// SIMATIC STEP 7 (V5.x) project Mangal
// CPU: CPU 416-2 DP
// station: Hardware
// station: SIMATIC 400
// station: P_ADR_BUS
// program: S7 Program(1)

SYMBOL_TABLE
"CONT_C"	FB 1	FB 1	// Continuous PID controller
"TIMER_P"	FB 5	FB 5	// Impulsefunction and delayed On/Off
"RAMP_P"	FB 52	FB 52
"N_PID"	FB 55	FB 55
"regulator"	FB 321	FB 321
"CBCTRLS1"	FB 945	FB 945	// CB SEND DATA 1 TO CTR
"VISU_IND_CODE"	FB 982	FB 982	// VISU COLOR INDICATION CODE
"READY_STD"	FB 1060	FB 1060	// Diagnosis  block
"VISU_GEN"	FB 1067	FB 1067	// Visualisierung for general Indications
"N_AnMeas"	FB 1435	FB 1435
"N_SPMANIP"	FB 1467	FB 1467
"N_TON"	FB 1482	FB 1482
"N_TOF"	FB 1483	FB 1483
"CUT_SHER"	FB 3333	FB 3333
"A_IN"	FC 402	FC 402	// Analog Input Driver
"N_AW_BO"	FC 430	FC 430
"CYCL_EXC"	OB 1	OB 1	// Cycle Execution
"PROG_ERR"	OB 121	OB 121	// Programming Error
"MOD_ERR"	OB 122	OB 122	// Module Access Error
"TON"	SFB 4	SFB 4	// Generate an On Delay
"TOF"	SFB 5	SFB 5	// Generate an Off Delay
"ALARM_8P"	SFB 35	SFB 35	// Generate Block-Related Messages with Values for 8 Signals
"RD_SINFO"	SFC 6	SFC 6	// Read OB Start Information
"BLKMOV"	SFC 20	SFC 20	// Copy Variables
"TIME_TCK"	SFC 64	SFC 64	// Read the System Time
END_SYMBOL_TABLE

FUNCTION_BLOCK "CONT_C"	// FB 1
TITLE = Continuous PID controller
AUTHOR : ELEM_400
FAMILY : CONTROL
NAME : CONT_C
VERSION : 1.5
VAR_INPUT
  MAN_ON : BOOL  := TRUE;	//Select: 1=Manual Value, 0= Manip. Value
  PVPER_ON { S7_visible := 'false' }: BOOL ;	//Enable: 1=Process var. to Peripherl Dev.
  P_SEL : BOOL  := TRUE;	//1=Proportional Action ON
  I_SEL : BOOL  := TRUE;	//Enable: 1=Integral Action ON
  INT_HOLD : BOOL ;	//Integral Action Hold
  I_ITL_ON : BOOL ;	//Initialize Integral Action
  D_SEL : BOOL ;	//1=Derivative Action ON
  SAMPLE_T { S7_visible := 'false'; S7_sampletime := 'true' }: REAL  := 1.000000e+000;	//Sample Time [s]
  SP_INT : REAL ;	//Internal setpoint
  PV_IN { S7_dynamic := 'true' }: REAL ;	//Process Variable Input
  PV_PER : WORD ;	//Process Variable from Peripheral Device
  MAN : REAL ;	//Operator Entered Manual Value
  GAIN { S7_dynamic := 'true'; S7_edit := 'para' }: REAL  := 2.000000e+000;	//Proportional Gain
  TN { S7_dynamic := 'true'; S7_edit := 'para' }: TIME  := T#20S;	//Reset time [sec]
  TV { S7_dynamic := 'true'; S7_edit := 'para' }: TIME  := T#10S;	//Differential Time [s]
  TM_LAG : TIME  := T#2S;	//Lag Time of the Derivative Action [sec]
  DEADB_W : REAL ;	//Deadband width
  LMN_HLM : REAL  := 1.000000e+002;	//Manipulated Value High Limit
  LMN_LLM : REAL ;	//Manipulated Value Low Limit
  PV_FAC { S7_visible := 'false' }: REAL  := 1.000000e+000;	//Process Variable Adjustment Factor
  PV_OFF { S7_visible := 'false' }: REAL ;	//Process Variable Offset
  LMN_FAC : REAL  := 1.000000e+000;	//Manipulated Value Adjustment Factor
  LMN_OFF : REAL ;	//Manipulated Value Offset
  I_ITLVAL : REAL ;	//Initialization Value of Integral Action
  DISV : REAL ;	//Disturbance variable
END_VAR
VAR_OUTPUT
  LMN : REAL ;	//Manipulated Value
  LMN_PER : WORD ;	//Manipulated Value for Peripheral Device
  QLMN_HLM : BOOL ;	//1=High Limit of Manipulated Value active
  QLMN_LLM : BOOL ;	//1=Low Limit of Manipulated Value active
  LMN_P : REAL ;	//Proportionality Component
  LMN_I : REAL ;	//Integral Component
  LMN_D : REAL ;	//Derivative Component
  PV { S7_visible := 'false' }: REAL ;	//Process Variable
  ER : REAL ;	//Error Signal
END_VAR
VAR
  sInvAlt : REAL ;
  sIanteilAlt : REAL ;
  sRestInt : REAL ;
  sRestDif : REAL ;
  sRueck : REAL ;
  sLmn : REAL ;
  sbArwHLmOn : BOOL ;
  sbArwLLmOn : BOOL ;
  sbILimOn : BOOL  := TRUE;
END_VAR
VAR_TEMP
  ERR : INT ;
  TOP_SI : STRUCT
   EV_CLASS : BYTE ;
   EV_NUM : BYTE ;
   PRIORITY : BYTE ;
   NUM : BYTE ;
   TYP2_3 : BYTE ;
   TYP1 : BYTE ;
   ZI1 : WORD ;
   ZI2_3 : DWORD ;
  END_STRUCT ;
  START_UP_SI : STRUCT
   EV_CLASS : BYTE ;
   EV_NUM : BYTE ;
   PRIORITY : BYTE ;
   NUM : BYTE ;
   TYP2_3 : BYTE ;
   TYP1 : BYTE ;
   ZI1 : WORD ;
   ZI2_3 : DWORD ;
  END_STRUCT ;
  Hvar : REAL ;	//Hilfsvariable
  Diff : REAL ;	//Änderungswert
  Istwert : REAL ;	//Istwert
  ErKp : REAL ;	//Hilfsvariable
  rTi : REAL ;	//Integrationszeit in real
  rTd : REAL ;	//Differentiationszeit in real
  rTmLag : REAL ;	//Verzögerungszeit in real
  Panteil : REAL ;	//P-Anteil
  Ianteil : REAL ;	//I-Anteil
  Danteil : REAL ;	//D-Anteil
  Verstaerk : REAL ;	//Verstärkung
  RueckDiff : REAL ;	//Differenz des Rückkopplungswertes
  RueckAlt : REAL ;	//Alter Rückkopplungswert
  dLmn : REAL ;	//Stellwert
  gf : REAL ;	//Hilfwert
  rVal : REAL ;	//Real Hilfsvariable
END_VAR
BEGIN
// body was compiled from an SCL source; compiled code not shown
END_FUNCTION_BLOCK

// FB 5: know-how protected block, not included

FUNCTION_BLOCK FB 45
VERSION : 0.1
BEGIN
// (block stored without names or comments; labels and parameter names are numbered)
END_FUNCTION_BLOCK

FUNCTION_BLOCK "RAMP_P"	// FB 52
TITLE = Rampforming
AUTHOR : BASIS70
FAMILY : CONTROL
NAME : RAMP_P
VERSION : 3.0
VAR_INPUT
  SAMPLE_T { S7_visible := 'false'; S7_sampletime := 'true' }: REAL  := 1.000000e+000;	//Sample Time [s]
  URLM { S7_dynamic := 'true'; S7_edit := 'para' }: REAL  := 3.000000e+000;	//Positive Ramp Rate Limit Output Value
  DRLM { S7_dynamic := 'true'; S7_edit := 'para' }: REAL  := 3.000000e+000;	//Max. negative Ramp Rate of Output Value
  U { S7_dynamic := 'true' }: REAL ;	//Input Value
  RATE_OFF { S7_dynamic := 'true' }: BOOL ;	//1=Ramp Rate Monitoring off
END_VAR
VAR_OUTPUT
  QERR { S7_visible := 'false' }: BOOL  := TRUE;	//1=Error
  QLIM_U { S7_dynamic := 'true' }: BOOL ;	//1=Positiv Ramp Rate Limit Active
  QLIM_D { S7_dynamic := 'true' }: BOOL ;	//1=Negativ Ramp Rate Limit Active
  V { S7_dynamic := 'true' }: REAL ;	//Analog Output
END_VAR
VAR
  srSAMPLE_T : REAL ;	//interne Abtastzeit
END_VAR
VAR_TEMP
  tbQlim_u : BOOL ;	//Hilfsmerker positiver Gradient zu gross
  tbQlim_d : BOOL ;	//Hilfsmerker negativer Gradient zu gross
  trGrad : REAL ;	//Gradient
  trDiff : REAL ;	//temporäre Var. für U-V
  ERR : INT ;	//Error beim Anlauf
  TOP_SI : STRUCT
   EV_CLASS : BYTE ;
   EV_NUM : BYTE ;
   PRIORITY : BYTE ;
   NUM : BYTE ;
   TYP2_3 : BYTE ;
   TYP1 : BYTE ;
   ZI1 : WORD ;
   ZI2_3 : DWORD ;
  END_STRUCT ;
  START_UP_SI : STRUCT
   EV_CLASS : BYTE ;
   EV_NUM : BYTE ;
   PRIORITY : BYTE ;
   NUM : BYTE ;
   TYP2_3 : BYTE ;
   TYP1 : BYTE ;
   ZI1 : WORD ;
   ZI2_3 : DWORD ;
  END_STRUCT ;
END_VAR
BEGIN
// body was compiled from an SCL source; compiled code not shown
END_FUNCTION_BLOCK

FUNCTION_BLOCK "N_PID"	// FB 55
VERSION : 0.1
VAR_INPUT
  PLCAUTOSP : BOOL ;
  PLCMANSP : BOOL ;
  PLCAUTOPOS : BOOL ;
  PLCMANPOS : BOOL ;
  P_SEL { S7_m_c := 'true' }: BOOL ;
  I_SEL { S7_m_c := 'true' }: BOOL ;
  D_SEL { S7_m_c := 'true' }: BOOL ;
  INT_HOLD : BOOL ;
  INT_INIT : BOOL ;
  SPAUTO { S7_m_c := 'true' }: REAL ;
  SPAUTOPOS { S7_m_c := 'true' }: REAL ;
  PV { S7_m_c := 'true' }: REAL ;
  GAIN { S7_m_c := 'true'; S7_dynamic := 'true' }: REAL ;
  TN { S7_dynamic := 'true'; S7_m_c := 'true' }: REAL ;
  TV { S7_dynamic := 'true'; S7_m_c := 'true' }: REAL ;
  TM_LAG : REAL ;
  DEAD_W : REAL ;
  DEV { S7_dynamic := 'true'; S7_m_c := 'true' }: REAL ;
  DEV_TIME { S7_dynamic := 'true'; S7_m_c := 'true' }: REAL ;	//Deviation time [s]
  LNM_HLIM : REAL ;
  LNM_LLIM : REAL ;
  I_INITVAL : REAL ;
  DISV : REAL ;
  SAMPLE_T { S7_sampletime := 'true' }: REAL ;
END_VAR
VAR_OUTPUT
  QAUTOSP { S7_dynamic := 'true'; S7_m_c := 'true' }: BOOL ;
  QMANSP { S7_dynamic := 'true'; S7_m_c := 'true' }: BOOL ;
  QAUTOPOS { S7_dynamic := 'true'; S7_m_c := 'true' }: BOOL ;
  QMANPOS { S7_dynamic := 'true'; S7_m_c := 'true' }: BOOL ;
  QLMN { S7_dynamic := 'true'; S7_m_c := 'true' }: REAL ;
  QLMN_P : REAL ;
  QLMN_I : REAL ;
  QLMN_D : REAL ;
  QLMN_HLIM : BOOL ;
  QLMM_LLIM : BOOL ;
  QDEV_H { S7_m_c := 'true' }: BOOL ;
  QDEV_L { S7_m_c := 'true' }: BOOL ;
  QDEV : BOOL ;
  QDEV_ACT : REAL ;
  QPID_SP { S7_dynamic := 'true'; S7_m_c := 'true' }: REAL ;
  QER { S7_dynamic := 'true'; S7_m_c := 'true' }: REAL ;
END_VAR
VAR_IN_OUT
  HMIAUTOSP { S7_dynamic := 'true'; S7_m_c := 'true' }: BOOL ;
  HMIMANSP { S7_dynamic := 'true'; S7_m_c := 'true' }: BOOL ;
  HMIAUTOPOS { S7_dynamic := 'true'; S7_m_c := 'true' }: BOOL ;
  HMIMANPOS { S7_dynamic := 'true'; S7_m_c := 'true' }: BOOL ;
  HMISPMAN { S7_dynamic := 'true'; S7_m_c := 'true' }: REAL ;
  HMISPMANPOS { S7_dynamic := 'true'; S7_m_c := 'true' }: REAL ;
  HMIOPEN { S7_m_c := 'true' }: BOOL ;
  HMICLOSE { S7_m_c := 'true' }: BOOL ;
END_VAR
VAR
  AutoSPMode_Int : BOOL ;
  AutoPosMode_Int : BOOL ;
  ManSPMode_Int : BOOL ;
  ManPosMode_Int : BOOL ;
  Pos : BOOL ;
  Reg : BOOL ;
  Deviation : BOOL ;
  Dev_H : BOOL ;
  Dev_L : BOOL ;
  HMIAtuoSPReq : BOOL ;
  HMIManSPReq : BOOL ;
  HMIAtuoPosReq : BOOL ;
  HMIManPosReq : BOOL ;
  ReqAutoSP : BOOL ;
  ReqManSP : BOOL ;
  ReqAutoPos : BOOL ;
  ReqManPos : BOOL ;
  PulsePLCAutoSP : BOOL ;
  PulsePLCManSP : BOOL ;
  PulsePLCAutoPos : BOOL ;
  PulsePLCManPos : BOOL ;
  Spare_11 : BOOL ;
  Spare_10 : BOOL ;
  Spare_9 : BOOL ;
  Spare_8 : BOOL ;
  Spare_7 : BOOL ;
  Spare_6 : BOOL ;
  Spare_5 : BOOL ;
  Spare_4 : BOOL ;
  Spare_3 : BOOL ;
  Spare_2 : BOOL ;
  Spare_1 : BOOL ;
  Spare1 : REAL ;
  Spare2 : REAL ;
  Spare3 : REAL ;
  AutoSP_Int : REAL ;
  ManSP_Int : REAL ;
  AutoPosSP_Int : REAL ;
  ManPosSP_Int : REAL ;
  PID_SP : REAL ;
  PID_SP_Ramped : REAL ;
  PID_Pos_SP : REAL ;
  PID_Pos_SP_Ramped : REAL ;
  PID_LMN : REAL ;
  Err_Val : REAL ;
  Dev_Val_Abs : REAL ;
  DEV_Act_Int : REAL ;
  DEV_Proc : REAL ;
  Dev_Tmr : SFB 4;
  PID_CTRL : FB 1;
  SP_RAMP : FB 52;
  POS_RAMP : FB 52;
  MANIP_SP : FB 1467;
END_VAR
VAR_TEMP
  Log_1 : BOOL ;
  Log_0 : BOOL ;
  TN_Int : TIME ;
  TV_Int : TIME ;
  TM_LAG_Int : TIME ;
  Dev_Time_Int : TIME ;
  Temp_Real : REAL ;
  Dummy_S5 : BOOL ;
END_VAR
BEGIN
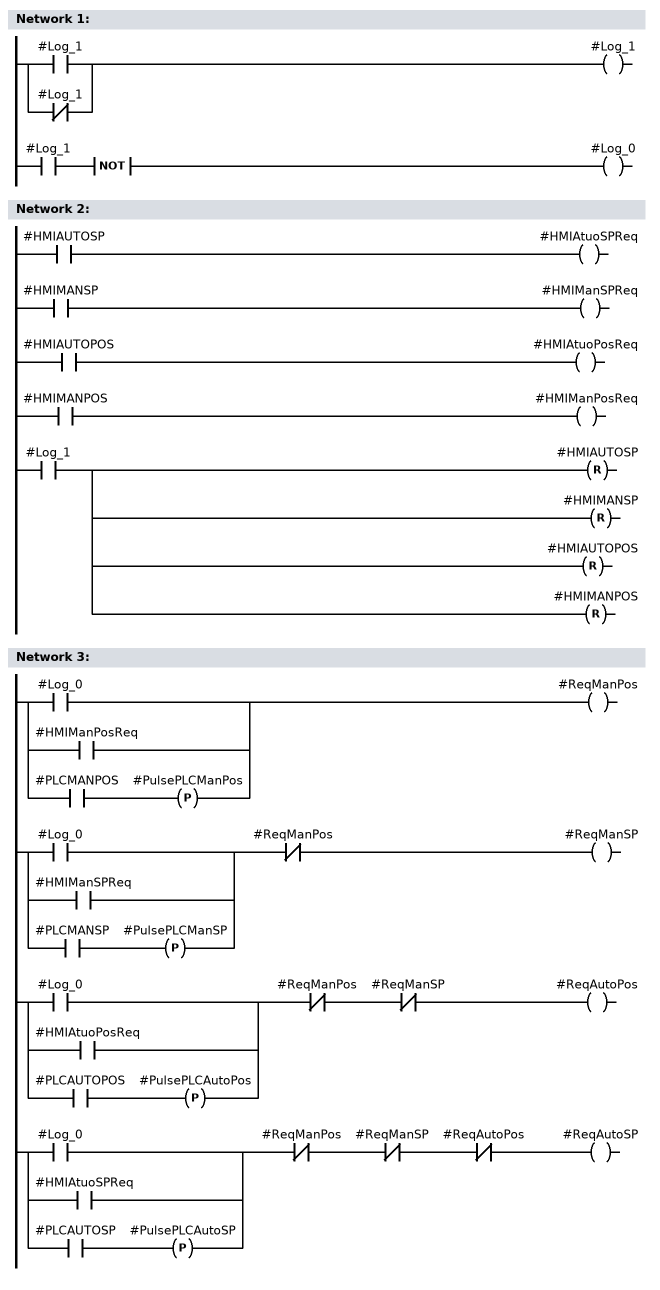
NETWORK
TITLE =
      A(;
      O     #Log_1;
      ON    #Log_1;
      );
      =     #Log_1;
      A     #Log_1;
      NOT;
      =     #Log_0;
NETWORK
TITLE =
      A     #HMIAUTOSP;
      =     #HMIAtuoSPReq;
      A     #HMIMANSP;
      =     #HMIManSPReq;
      A     #HMIAUTOPOS;
      =     #HMIAtuoPosReq;
      A     #HMIMANPOS;
      =     #HMIManPosReq;
      A     #Log_1;
      R     #HMIAUTOSP;
      R     #HMIMANSP;
      R     #HMIAUTOPOS;
      R     #HMIMANPOS;
NETWORK
TITLE =
      A     #Log_0;
      =     L 23.0;
      O     L 23.0;
      O     #HMIManPosReq;
      O(;
      A     #PLCMANPOS;
      FP    #PulsePLCManPos;
      );
      =     #ReqManPos;
      A(;
      O     L 23.0;
      O     #HMIManSPReq;
      O(;
      A     #PLCMANSP;
      FP    #PulsePLCManSP;
      );
      );
      AN    #ReqManPos;
      =     #ReqManSP;
      A(;
      O     L 23.0;
      O     #HMIAtuoPosReq;
      O(;
      A     #PLCAUTOPOS;
      FP    #PulsePLCAutoPos;
      );
      );
      AN    #ReqManPos;
      AN    #ReqManSP;
      =     #ReqAutoPos;
      A(;
      O     L 23.0;
      O     #HMIAtuoSPReq;
      O(;
      A     #PLCAUTOSP;
      FP    #PulsePLCAutoSP;
      );
      );
      AN    #ReqManPos;
      AN    #ReqManSP;
      AN    #ReqAutoPos;
      =     #ReqAutoSP;
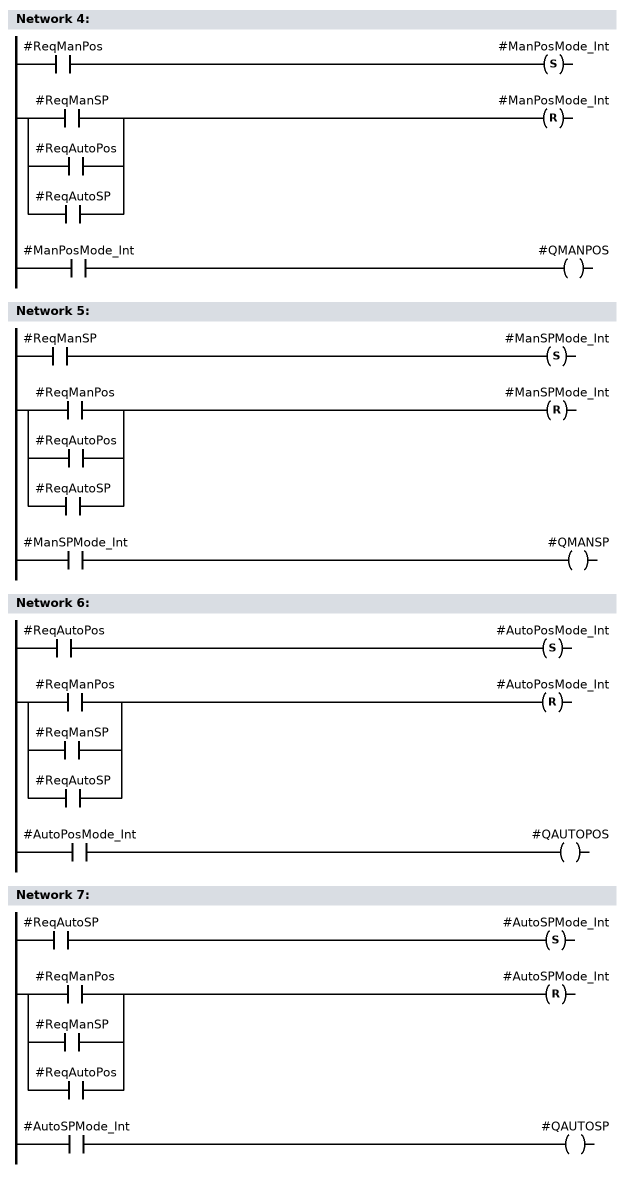
NETWORK
TITLE =
      A     #ReqManPos;
      S     #ManPosMode_Int;
      A(;
      O     #ReqManSP;
      O     #ReqAutoPos;
      O     #ReqAutoSP;
      );
      R     #ManPosMode_Int;
      A     #ManPosMode_Int;
      =     #QMANPOS;
NETWORK
TITLE =
      A     #ReqManSP;
      S     #ManSPMode_Int;
      A(;
      O     #ReqManPos;
      O     #ReqAutoPos;
      O     #ReqAutoSP;
      );
      R     #ManSPMode_Int;
      A     #ManSPMode_Int;
      =     #QMANSP;
NETWORK
TITLE =
      A     #ReqAutoPos;
      S     #AutoPosMode_Int;
      A(;
      O     #ReqManPos;
      O     #ReqManSP;
      O     #ReqAutoSP;
      );
      R     #AutoPosMode_Int;
      A     #AutoPosMode_Int;
      =     #QAUTOPOS;
NETWORK
TITLE =
      A     #ReqAutoSP;
      S     #AutoSPMode_Int;
      A(;
      O     #ReqManPos;
      O     #ReqManSP;
      O     #ReqAutoPos;
      );
      R     #AutoSPMode_Int;
      A     #AutoSPMode_Int;
      =     #QAUTOSP;
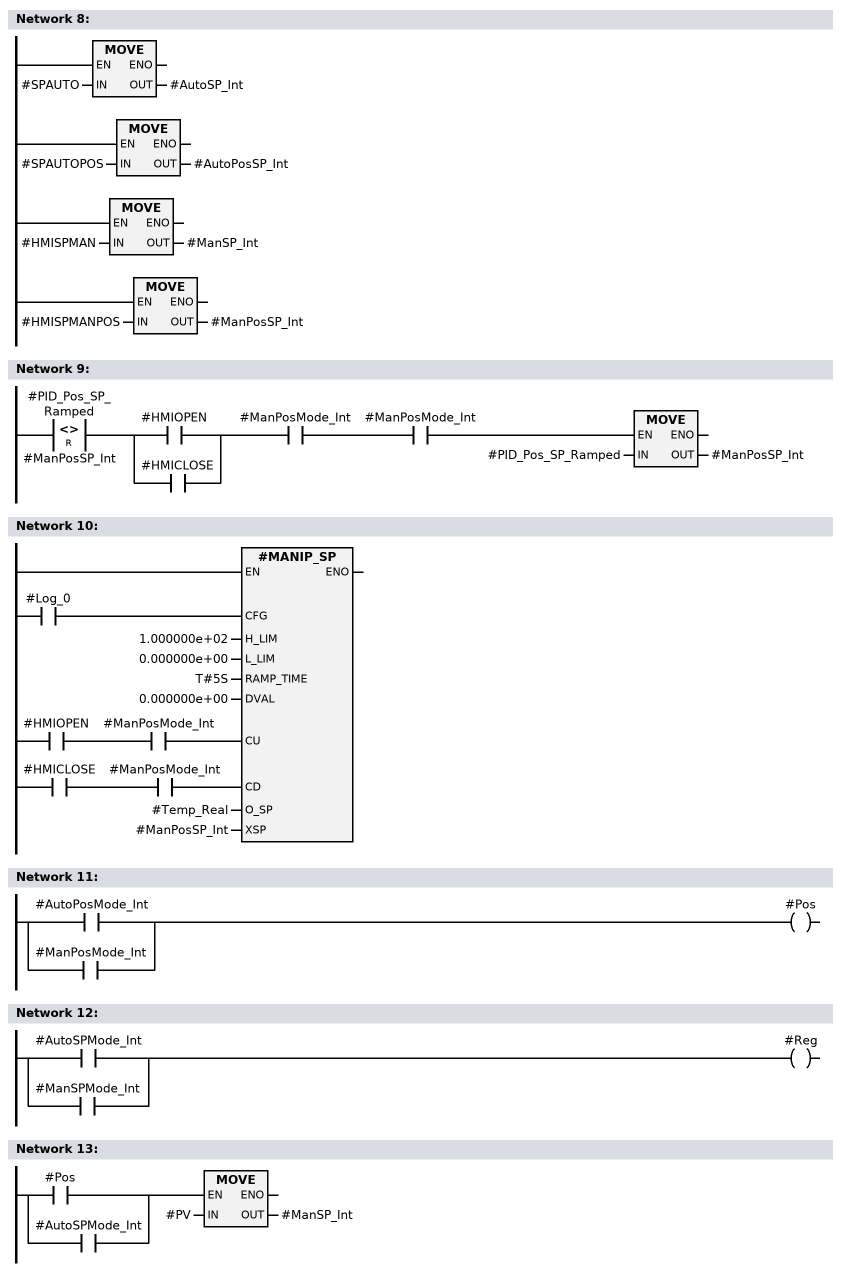
NETWORK
TITLE =
      L     #SPAUTO;
      T     #AutoSP_Int;
      L     #SPAUTOPOS;
      T     #AutoPosSP_Int;
      L     #HMISPMAN;
      T     #ManSP_Int;
      L     #HMISPMANPOS;
      T     #ManPosSP_Int;
NETWORK
TITLE =
      A(;
      L     #PID_Pos_SP_Ramped;
      L     #ManPosSP_Int;
      <>R;
      );
      A(;
      O     #HMIOPEN;
      O     #HMICLOSE;
      );
      A     #ManPosMode_Int;
      A     #ManPosMode_Int;
      JNB   _010;
      L     #PID_Pos_SP_Ramped;
      T     #ManPosSP_Int;
_010: NOP   0;
NETWORK
TITLE =
      A     #Log_0;
      =     L 23.0;
      BLD   103;
      A     #HMIOPEN;
      A     #ManPosMode_Int;
      =     L 23.3;
      BLD   103;
      A     #HMICLOSE;
      A     #ManPosMode_Int;
      =     L 23.4;
      BLD   103;
      CALL  #MANIP_SP (
           CFG                      := L 23.0,
           H_LIM                    := 1.000000e+02,
           L_LIM                    := 0.000000e+00,
           RAMP_TIME                := T#5S,
           DVAL                     := 0.000000e+00,
           CU                       := L 23.3,
           CD                       := L 23.4,
           O_SP                     := #Temp_Real,
           XSP                      := #ManPosSP_Int);
      NOP   0;
NETWORK
TITLE =
      O     #AutoPosMode_Int;
      O     #ManPosMode_Int;
      =     #Pos;
NETWORK
TITLE =
      O     #AutoSPMode_Int;
      O     #ManSPMode_Int;
      =     #Reg;
NETWORK
TITLE =
      A(;
      O     #Pos;
      O     #AutoSPMode_Int;
      );
      JNB   _011;
      L     #PV;
      T     #ManSP_Int;
_011: NOP   0;
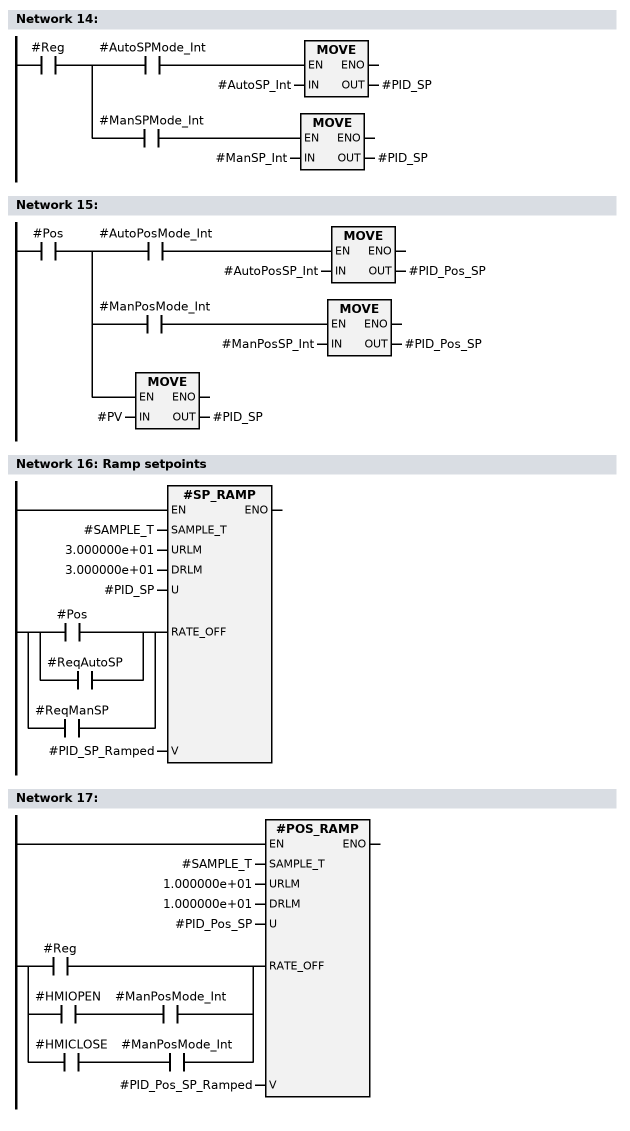
NETWORK
TITLE =
      A     #Reg;
      =     L 23.0;
      A     L 23.0;
      A     #AutoSPMode_Int;
      JNB   _012;
      L     #AutoSP_Int;
      T     #PID_SP;
_012: NOP   0;
      A     L 23.0;
      A     #ManSPMode_Int;
      JNB   _013;
      L     #ManSP_Int;
      T     #PID_SP;
_013: NOP   0;
NETWORK
TITLE =
      A     #Pos;
      =     L 23.0;
      A     L 23.0;
      A     #AutoPosMode_Int;
      JNB   _014;
      L     #AutoPosSP_Int;
      T     #PID_Pos_SP;
_014: NOP   0;
      A     L 23.0;
      A     #ManPosMode_Int;
      JNB   _015;
      L     #ManPosSP_Int;
      T     #PID_Pos_SP;
_015: NOP   0;
      A     L 23.0;
      JNB   _016;
      L     #PV;
      T     #PID_SP;
_016: NOP   0;
NETWORK
TITLE = Ramp setpoints
      A(;
      O     #Pos;
      O     #ReqAutoSP;
      O     #ReqManSP;
      );
      =     L 23.0;
      BLD   103;
      CALL  #SP_RAMP (
           SAMPLE_T                 := #SAMPLE_T,
           URLM                     := 3.000000e+01,
           DRLM                     := 3.000000e+01,
           U                        := #PID_SP,
           RATE_OFF                 := L 23.0,
           V                        := #PID_SP_Ramped);
      NOP   0;
NETWORK
TITLE =
      A(;
      O     #Reg;
      O;
      A     #HMIOPEN;
      A     #ManPosMode_Int;
      O;
      A     #HMICLOSE;
      A     #ManPosMode_Int;
      );
      =     L 23.0;
      BLD   103;
      CALL  #POS_RAMP (
           SAMPLE_T                 := #SAMPLE_T,
           URLM                     := 1.000000e+01,
           DRLM                     := 1.000000e+01,
           U                        := #PID_Pos_SP,
           RATE_OFF                 := L 23.0,
           V                        := #PID_Pos_SP_Ramped);
      NOP   0;
NETWORK
TITLE = Real to TIME conversion
      L     #TN;
      L     1.000000e+03;
      *R;
      RND;
      T     #TN_Int;
      L     #TV;
      L     1.000000e+03;
      *R;
      RND;
      T     #TV_Int;
      L     #TM_LAG;
      L     1.000000e+03;
      *R;
      RND;
      T     #TM_LAG_Int;
      L     #DEV_TIME;
      L     1.000000e+03;
      *R;
      RND;
      T     #Dev_Time_Int;
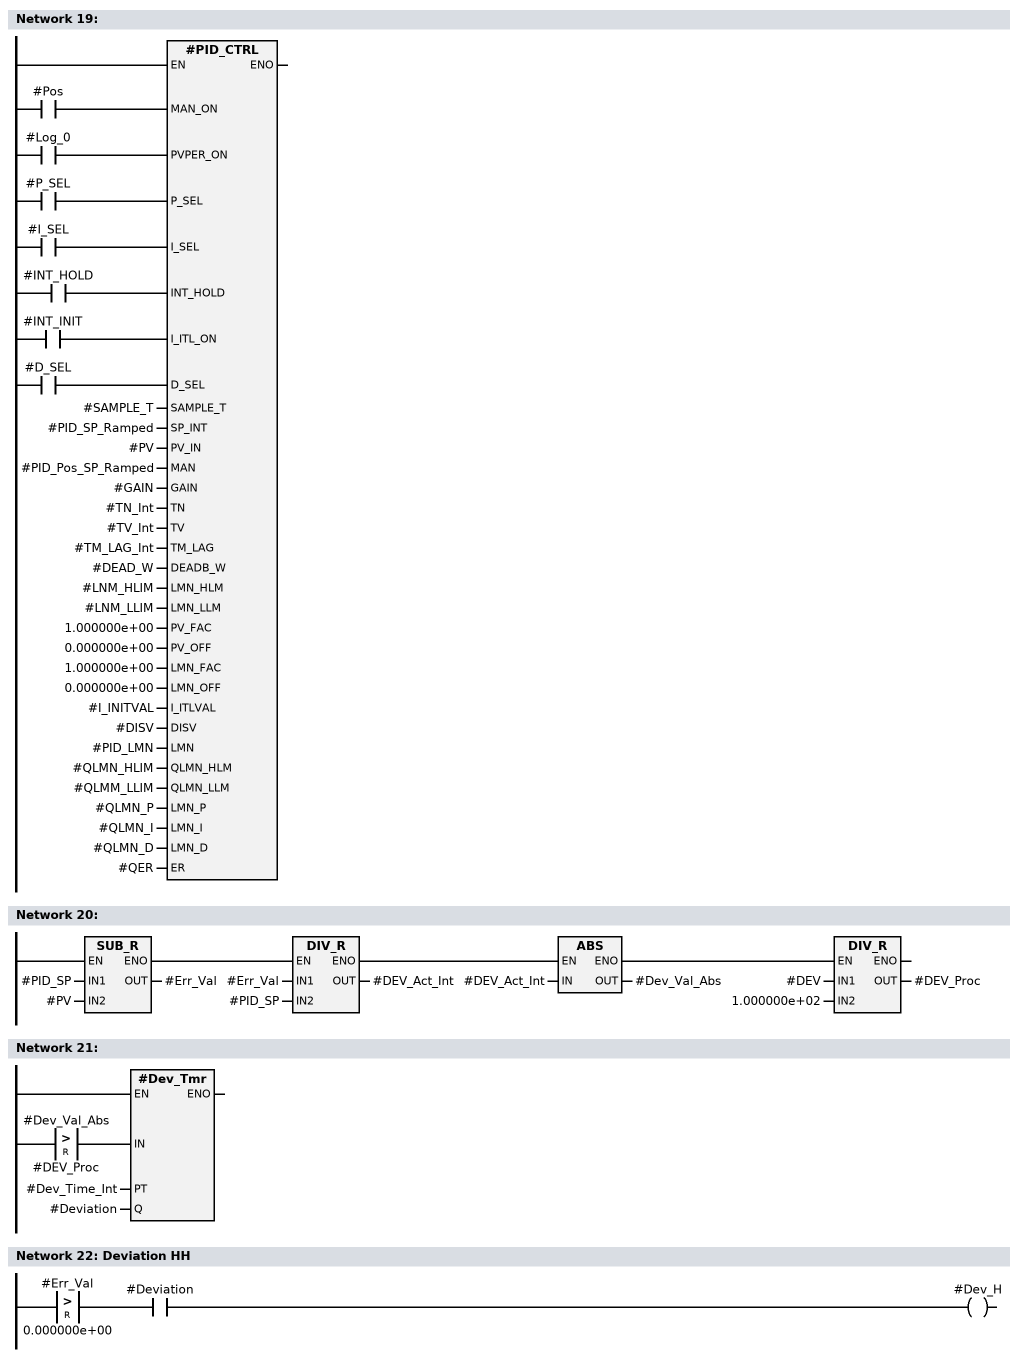
NETWORK
TITLE =
      A     #Pos;
      =     L 23.0;
      BLD   103;
      A     #Log_0;
      =     L 23.1;
      BLD   103;
      A     #P_SEL;
      =     L 23.2;
      BLD   103;
      A     #I_SEL;
      =     L 23.3;
      BLD   103;
      A     #INT_HOLD;
      =     L 23.4;
      BLD   103;
      A     #INT_INIT;
      =     L 23.5;
      BLD   103;
      A     #D_SEL;
      =     L 23.6;
      BLD   103;
      CALL  #PID_CTRL (
           MAN_ON                   := L 23.0,
           PVPER_ON                 := L 23.1,
           P_SEL                    := L 23.2,
           I_SEL                    := L 23.3,
           INT_HOLD                 := L 23.4,
           I_ITL_ON                 := L 23.5,
           D_SEL                    := L 23.6,
           SAMPLE_T                 := #SAMPLE_T,
           SP_INT                   := #PID_SP_Ramped,
           PV_IN                    := #PV,
           MAN                      := #PID_Pos_SP_Ramped,
           GAIN                     := #GAIN,
           TN                       := #TN_Int,
           TV                       := #TV_Int,
           TM_LAG                   := #TM_LAG_Int,
           DEADB_W                  := #DEAD_W,
           LMN_HLM                  := #LNM_HLIM,
           LMN_LLM                  := #LNM_LLIM,
           PV_FAC                   := 1.000000e+00,
           PV_OFF                   := 0.000000e+00,
           LMN_FAC                  := 1.000000e+00,
           LMN_OFF                  := 0.000000e+00,
           I_ITLVAL                 := #I_INITVAL,
           DISV                     := #DISV,
           LMN                      := #PID_LMN,
           QLMN_HLM                 := #QLMN_HLIM,
           QLMN_LLM                 := #QLMM_LLIM,
           LMN_P                    := #QLMN_P,
           LMN_I                    := #QLMN_I,
           LMN_D                    := #QLMN_D,
           ER                       := #QER);
      NOP   0;
NETWORK
TITLE =
      A(;
      A(;
      A(;
      L     #PID_SP;
      L     #PV;
      -R;
      T     #Err_Val;
      AN    OV;
      SAVE;
      CLR;
      A     BR;
      );
      JNB   _017;
      L     #Err_Val;
      L     #PID_SP;
      /R;
      T     #DEV_Act_Int;
      AN    OV;
      SAVE;
      CLR;
_017: A     BR;
      );
      JNB   _01c;
      L     #DEV_Act_Int;
      ABS;
      T     #Dev_Val_Abs;
      SET;
      SAVE;
      CLR;
_01c: A     BR;
      );
      JNB   _01d;
      L     #DEV;
      L     1.000000e+02;
      /R;
      T     #DEV_Proc;
_01d: NOP   0;
NETWORK
TITLE =
      A(;
      L     #Dev_Val_Abs;
      L     #DEV_Proc;
      >R;
      );
      =     L 23.0;
      BLD   103;
      CALL  #Dev_Tmr (
           IN                       := L 23.0,
           PT                       := #Dev_Time_Int,
           Q                        := #Deviation);
      NOP   0;
NETWORK
TITLE = Deviation HH
      A(;
      L     #Err_Val;
      L     0.000000e+00;
      >R;
      );
      A     #Deviation;
      =     #Dev_H;
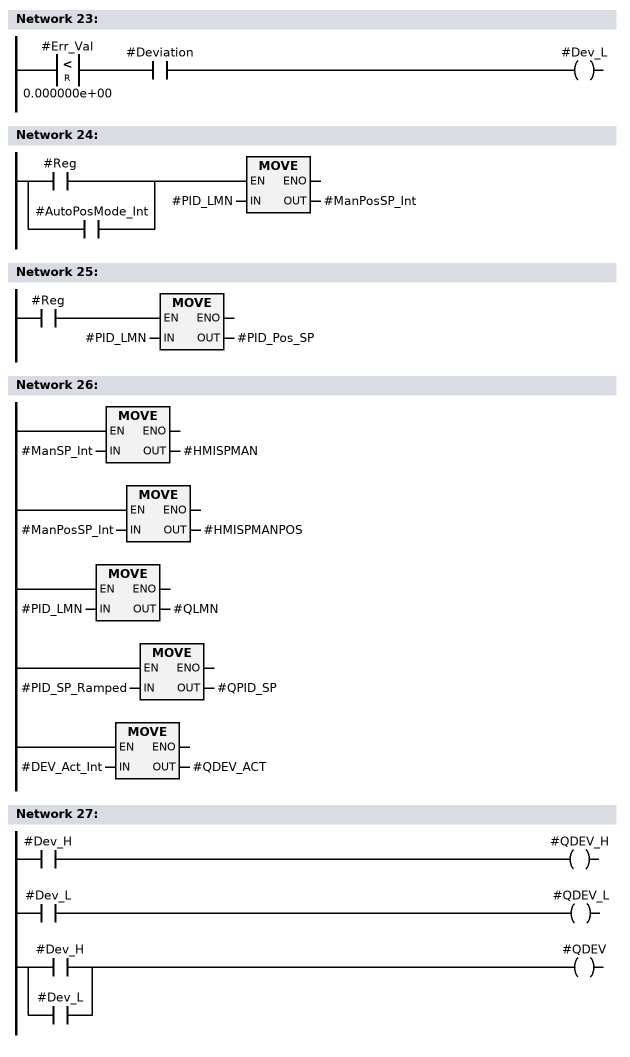
NETWORK
TITLE =
      A(;
      L     #Err_Val;
      L     0.000000e+00;
      <R;
      );
      A     #Deviation;
      =     #Dev_L;
NETWORK
TITLE =
      A(;
      O     #Reg;
      O     #AutoPosMode_Int;
      );
      JNB   _01e;
      L     #PID_LMN;
      T     #ManPosSP_Int;
_01e: NOP   0;
NETWORK
TITLE =
      A     #Reg;
      JNB   _01f;
      L     #PID_LMN;
      T     #PID_Pos_SP;
_01f: NOP   0;
NETWORK
TITLE =
      L     #ManSP_Int;
      T     #HMISPMAN;
      L     #ManPosSP_Int;
      T     #HMISPMANPOS;
      L     #PID_LMN;
      T     #QLMN;
      L     #PID_SP_Ramped;
      T     #QPID_SP;
      L     #DEV_Act_Int;
      T     #QDEV_ACT;
NETWORK
TITLE =
      A     #Dev_H;
      =     #QDEV_H;
      A     #Dev_L;
      =     #QDEV_L;
      A     #Dev_H;
      O     #Dev_L;
      =     #QDEV;
END_FUNCTION_BLOCK

FUNCTION_BLOCK "regulator"	// FB 321
VERSION : 0.1
VAR_INPUT
  SENSOR : REAL ;
  REF_OPERATOR : REAL ;
  LIMIT_UP : REAL ;
  LIMIT_DOWN : REAL ;
  VA_UP : REAL ;
  REFOR : REAL ;
  HW_PULS : BOOL ;
END_VAR
VAR_OUTPUT
  OUT_HEX : REAL ;
  OPEN_VALVE : BOOL ;
  CLOSET_VALVE : BOOL ;
END_VAR
VAR
  PERSENT : REAL ;
  DOLA_UP_1 : REAL ;
  DOLA_UP : REAL ;
  ALL_REF_UP : REAL ;
  ALL_REF_DOWN : REAL ;
  REFFF : REAL ;
  BIT_1 : BOOL ;
  BIT_2 : BOOL ;
  STOP_UP : BOOL ;
  STOP_DOWN : BOOL ;
END_VAR
BEGIN
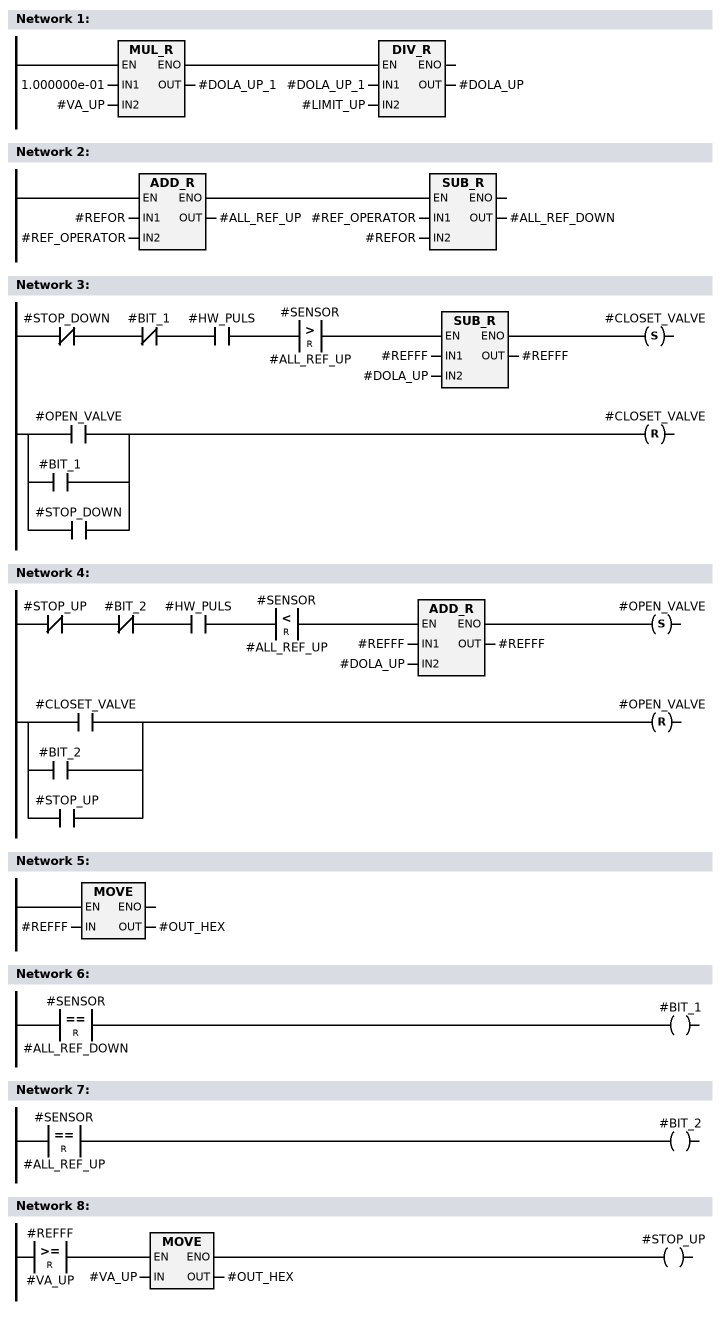
NETWORK
TITLE =
      A(;
      L     1.000000e-01;
      L     #VA_UP;
      *R;
      T     #DOLA_UP_1;
      AN    OV;
      SAVE;
      CLR;
      A     BR;
      );
      JNB   _001;
      L     #DOLA_UP_1;
      L     #LIMIT_UP;
      /R;
      T     #DOLA_UP;
_001: NOP   0;
NETWORK
TITLE =
      A(;
      L     #REFOR;
      L     #REF_OPERATOR;
      +R;
      T     #ALL_REF_UP;
      AN    OV;
      SAVE;
      CLR;
      A     BR;
      );
      JNB   _002;
      L     #REF_OPERATOR;
      L     #REFOR;
      -R;
      T     #ALL_REF_DOWN;
_002: NOP   0;
NETWORK
TITLE =
      A(;
      AN    #STOP_DOWN;
      AN    #BIT_1;
      A     #HW_PULS;
      A(;
      L     #SENSOR;
      L     #ALL_REF_UP;
      >R;
      );
      JNB   _003;
      L     #REFFF;
      L     #DOLA_UP;
      -R;
      T     #REFFF;
      AN    OV;
      SAVE;
      CLR;
_003: A     BR;
      );
      S     #CLOSET_VALVE;
      A(;
      O     #OPEN_VALVE;
      O     #BIT_1;
      O     #STOP_DOWN;
      );
      R     #CLOSET_VALVE;
      NOP   0;
NETWORK
TITLE =
      A(;
      AN    #STOP_UP;
      AN    #BIT_2;
      A     #HW_PULS;
      A(;
      L     #SENSOR;
      L     #ALL_REF_UP;
      <R;
      );
      JNB   _004;
      L     #REFFF;
      L     #DOLA_UP;
      +R;
      T     #REFFF;
      AN    OV;
      SAVE;
      CLR;
_004: A     BR;
      );
      S     #OPEN_VALVE;
      A(;
      O     #CLOSET_VALVE;
      O     #BIT_2;
      O     #STOP_UP;
      );
      R     #OPEN_VALVE;
      NOP   0;
NETWORK
TITLE =
      L     #REFFF;
      T     #OUT_HEX;
      NOP   0;
NETWORK
TITLE =
      L     #SENSOR;
      L     #ALL_REF_DOWN;
      ==R;
      =     #BIT_1;
NETWORK
TITLE =
      L     #SENSOR;
      L     #ALL_REF_UP;
      ==R;
      =     #BIT_2;
NETWORK
TITLE =
      A(;
      L     #REFFF;
      L     #VA_UP;
      >=R;
      );
      JNB   _005;
      L     #VA_UP;
      T     #OUT_HEX;
      SET;
      SAVE;
      CLR;
_005: A     BR;
      =     #STOP_UP;
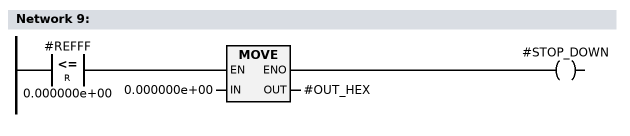
NETWORK
TITLE =
      A(;
      L     #REFFF;
      L     0.000000e+00;
      <=R;
      );
      JNB   _006;
      L     0.000000e+00;
      T     #OUT_HEX;
      SET;
      SAVE;
      CLR;
_006: A     BR;
      =     #STOP_DOWN;
END_FUNCTION_BLOCK

FUNCTION_BLOCK "CBCTRLS1"	// FB 945
TITLE = CB SEND DATA 1 TO CTR
//
//
//Create date: 11.08.1999        Date of last change: 28.01.2002
//
//Module for Bar and Rod Mills
//
//Module SB5COL11
//
//For more Details use online help
//
//Version V 5.01.00.00
//
//COPYRIGHT (C) SIEMENS AG 2001 ALL RIGHTS RESERVED
//
//
AUTHOR : SB5COL11
FAMILY : BRM_CCO
NAME : CBCTRLS1
VERSION : 1.8
VAR_INPUT
  SI_US { S7_m_c := 'false' }: INT ;	//0=SI, 1=US CUSTOMARY UNITS
  DBCTRLS : BLOCK_DB ;	//DB-NUMBER OF USED DATABLOCK
  XDISSND { S7_m_c := 'false' }: BOOL ;	//DISABLE: SEND PROCESS TO DB
END_VAR
VAR_OUTPUT
  YDISSND { S7_m_c := 'false' }: BOOL ;	//DISABLE: SEND PROCESS TO DB
END_VAR
VAR_IN_OUT
  COPMOFF { S7_m_c := 'false' }: BOOL ;	//CB: OPERATING MODE: OFF
  COPMMNT { S7_m_c := 'false' }: BOOL ;	//CB: OPERATING MODE: MAINTENANCE
  COPMLOC { S7_m_c := 'false' }: BOOL ;	//CB: OPERATING MODE: LOCAL
  COPMMAN { S7_m_c := 'false' }: BOOL ;	//CB: OPERATING MODE: MANUAL
  COPMAUT { S7_m_c := 'false' }: BOOL ;	//CB: OPERATING MODE: AUTOMATIC
  COPMSIM { S7_m_c := 'false' }: BOOL ;	//CB: OPERATING MODE: SIMULATION
  BITR6 { S7_m_c := 'false' }: BOOL ;	//CB: RESERVE
  COOLON { S7_m_c := 'false' }: BOOL ;	//CB: COOLING BED SETPOINT RELEASED
  ACK { S7_m_c := 'false' }: BOOL ;	//CB: FAULT ACKNOWLEDGE COOL AREA
  NSCHR { S7_m_c := 'false' }: BOOL ;	//CB: NEW SCHEDULE REACHED (PULSE)
  CLINEA { S7_m_c := 'false' }: BOOL ;	//CB: ROLLING LINE A ACTIVE
  CLINEB { S7_m_c := 'false' }: BOOL ;	//CB: ROLLING LINE B ACTIVE
  CLINEAB { S7_m_c := 'false' }: BOOL ;	//CB: ROLLING LINE AB ACTIVE
  BARON { S7_m_c := 'false' }: BOOL ;	//CB: BAR ROLLING ACTIVE TO CB
  R65 { S7_m_c := 'false' }: BOOL ;	//CB: RESERVE
  NOESTOP { S7_m_c := 'false' }: BOOL ;	//CB: NO ESTOP ACTIVATED
  FURSTOP { S7_m_c := 'false' }: BOOL ;	//CB: FURNACE STOP (DO NOT DISCHARGE)
  ROLSTOP { S7_m_c := 'false' }: BOOL ;	//CB: ROLLING STOP (AFTER TIME xx)
  CHOPP { S7_m_c := 'false' }: BOOL ;	//CB: CHOPPING COMMAND FROM COOL
  CBEMPTY { S7_m_c := 'false' }: BOOL ;	//CB: COOLING BED AREA EMPTY
  RDOPALL { S7_m_c := 'false' }: BOOL ;	//CB: READY FOR OPERATION ALL
  NOENTRY { S7_m_c := 'false' }: BOOL ;	//CB: NO ENTRY IN COOLING BED AREA
  ENBOP { S7_m_c := 'false' }: BOOL ;	//CB: ENTRY ENABLE OPERATOR
  R78 { S7_m_c := 'false' }: BOOL ;	//CB: RESERVE
  R79 { S7_m_c := 'false' }: BOOL ;	//CB: RESERVE
  R80 { S7_m_c := 'false' }: BOOL ;	//CB: RESERVE
  R81 { S7_m_c := 'false' }: BOOL ;	//CB: RESERVE
  R82 { S7_m_c := 'false' }: BOOL ;	//CB: RESERVE
  R83 { S7_m_c := 'false' }: BOOL ;	//CB: RESERVE
  R84 { S7_m_c := 'false' }: BOOL ;	//CB: RESERVE
  R85 { S7_m_c := 'false' }: BOOL ;	//CB: RESERVE
  R86 { S7_m_c := 'false' }: BOOL ;	//CB: RESERVE
  R91 { S7_m_c := 'false' }: REAL ;	//CB: RESERVE
  R92 { S7_m_c := 'false' }: REAL ;	//CB: RESERVE
  R93 { S7_m_c := 'false' }: REAL ;	//CB: RESERVE
  R94 { S7_m_c := 'false' }: REAL ;	//CB: RESERVE
  R95 { S7_m_c := 'false' }: REAL ;	//CB: RESERVE
  R96 { S7_m_c := 'false' }: REAL ;	//CB: RESERVE
  R97 { S7_m_c := 'false' }: REAL ;	//CB: RESERVE
  R98 { S7_m_c := 'false' }: REAL ;	//CB: RESERVE
  R99 { S7_m_c := 'false' }: REAL ;	//CB: RESERVE
  R100 { S7_m_c := 'false' }: REAL ;	//CB: RESERVE
  R101 { S7_m_c := 'false' }: INT ;	//CB: RESERVE
  R102 { S7_m_c := 'false' }: INT ;	//CB: RESERVE
  R103 { S7_m_c := 'false' }: INT ;	//CB: RESERVE
  R104 { S7_m_c := 'false' }: INT ;	//CB: RESERVE
  R105 { S7_m_c := 'false' }: INT ;	//CB: RESERVE
  R106 { S7_m_c := 'false' }: INT ;	//CB: RESERVE
  R107 { S7_m_c := 'false' }: INT ;	//CB: RESERVE
  R108 { S7_m_c := 'false' }: INT ;	//CB: RESERVE
  R109 { S7_m_c := 'false' }: INT ;	//CB: RESERVE
  R110 { S7_m_c := 'false' }: INT ;	//CB: RESERVE
END_VAR
VAR
  FACT_MS : REAL ;	//FACTOR FOR [m/s] TO [ft/min]
  FACT_METER : REAL ;	//FACTOR FOR [m]   TO [ft]
  FACT_MM : REAL ;	//FACTOR FOR [mm]  TO [inch]
  FACT_CM : REAL ;	//FACTOR FOR [cm]  TO [inch]
  FACT_KG : REAL ;	//FACTOR FOR [kg]  TO [lb]
  FACT_KGM : REAL ;	//FACTOR FOR [kg/m]TO [lb/ft]
END_VAR
BEGIN
// body was compiled from an SCL source; compiled code not shown
END_FUNCTION_BLOCK

FUNCTION_BLOCK "VISU_IND_CODE"	// FB 982
AUTHOR : SLCI&SIP
FAMILY : SLCI&SIP
NAME : VISU_IND
VERSION : 0.1
VAR_INPUT
  GY : BOOL ;	//COLOR GRAY (0)
  RD : BOOL ;	//COLOR RED (1)
  DARK_GN : BOOL ;	//COLOR DARK GREEN (2)
  RD_WH : BOOL ;	//COLOR RED WHITE FLUSH (256)
  MG : BOOL ;	//COLOR MAGENDA (512)
  DIR1_YE : BOOL ;	//COLOR DIRECTION 1 YELLOW (4)
  DIR1_YE_WH : BOOL ;	//COLOR DIRECTION 1 YELLOW WHITE FLUSH (8)
  DIR1_GN : BOOL ;	//COLOR DIRECTION 1 GREEN (16)
  DIR1_GN_WH : BOOL ;	//COLOR DIRECTION 1 GREEN WHITE FLUSH (32)
  DIR1_BU : BOOL ;	//COLOR DIRECTION 1 BLUE (64)
  DIR1_BU_WH : BOOL ;	//COLOR DIRECTION 1 BLUE WHITE FLUSH(128)
  DIR2_YE : BOOL ;	//COLOR DIRECTION 2 YELLOW (1024)
  DIR2_YE_WH : BOOL ;	//COLOR DIRECTION 2 YELLOW WHITE FLUSH (2048)
  DIR2_GN : BOOL ;	//COLOR DIRECTION 2 GREEN (4096)
  DIR2_GN_WH : BOOL ;	//COLOR DIRECTION 2 GREEN WHITE FLUSH (8192)
  DIR2_BU : BOOL ;	//COLOR DIRECTION 2 BLUE (16384)
  DIR2_BU_WH : BOOL ;	//COLOR DIRECTION 2 BLUE WHITE FLUSH(32768)
END_VAR
VAR_OUTPUT
  STATE { S7_m_c := 'true' }: INT ;	//STATUS INDICATION
END_VAR
BEGIN
NETWORK
TITLE =
      AN    #GY;
      JC    M001;
      L     0;
      JU    OUT;
M001: AN    #RD;
      JC    M002;
      L     1;
      JU    OUT;
M002: AN    #DARK_GN;
      JC    M003;
      L     2;
      JU    OUT;
M003: AN    #RD_WH;
      JC    M004;
      L     256;
      JU    OUT;
M004: AN    #MG;
      JC    M005;
      L     512;
      JU    OUT;
M005: AN    #DIR1_YE;
      JC    M006;
      L     4;
      JU    OUT;
M006: AN    #DIR1_YE_WH;
      JC    M007;
      L     8;
      JU    OUT;
M007: AN    #DIR1_GN;
      JC    M008;
      L     16;
      JU    OUT;
M008: AN    #DIR1_GN_WH;
      JC    M009;
      L     32;
      JU    OUT;
M009: AN    #DIR1_BU;
      JC    M010;
      L     64;
      JU    OUT;
M010: AN    #DIR1_BU_WH;
      JC    M011;
      L     128;
      JU    OUT;
M011: AN    #DIR2_YE;
      JC    M012;
      L     1024;
      JU    OUT;
M012: AN    #DIR2_YE_WH;
      JC    M013;
      L     2048;
      JU    OUT;
M013: AN    #DIR2_GN;
      JC    M014;
      L     4096;
      JU    OUT;
M014: AN    #DIR2_GN_WH;
      JC    M015;
      L     8192;
      JU    OUT;
M015: AN    #DIR2_BU;
      JC    M016;
      L     16384;
      JU    OUT;
M016: AN    #DIR1_BU_WH;
      JC    M017;
      L     W#16#8000;
      JU    OUT;
M017: L     0;
OUT:  T     #STATE;
END_FUNCTION_BLOCK

FUNCTION_BLOCK "READY_STD"	// FB 1060
TITLE = Condition of stand
//CHANGE #1  : Neue TC-Bibliothek SB1BASE0 und SB1DRIV0 V07.06.00.00; mit PCS7 
//V6.1 übersetzt    19.12.05
//
AUTHOR : Siemens
FAMILY : Projects
NAME : STD_COND
VERSION : 0.1
VAR_INPUT
  FAULT_01 { S7_m_c := 'true' }: BOOL ;	//Fault reason 1
  FAULT_02 { S7_m_c := 'true' }: BOOL ;	//Fault reason 2
  FAULT_03 { S7_m_c := 'true' }: BOOL ;	//Fault reason 3
  FAULT_04 { S7_m_c := 'true' }: BOOL ;	//Fault reason 4
  FAULT_05 { S7_m_c := 'true' }: BOOL ;	//Fault reason 5
  FAULT_06 { S7_m_c := 'true' }: BOOL ;	//Fault reason 6
  FAULT_07 { S7_m_c := 'true' }: BOOL ;	//Fault reason 7
  FAULT_08 { S7_m_c := 'true' }: BOOL ;	//Fault reason 8
  FAULT_09 { S7_m_c := 'true' }: BOOL ;	//Fault reason 9
  FAULT_10 { S7_m_c := 'true' }: BOOL ;	//Fault reason 10
  FAULT_11 { S7_m_c := 'true' }: BOOL ;	//Fault reason 11
  FAULT_12 { S7_m_c := 'true' }: BOOL ;	//Fault reason 12
  FAULT_13 { S7_m_c := 'true' }: BOOL ;	//Fault reason 13
  FAULT_14 { S7_m_c := 'true' }: BOOL ;	//Fault reason 14
  FAULT_15 { S7_m_c := 'true' }: BOOL ;	//Fault reason 15
  FAULT_16 { S7_m_c := 'true' }: BOOL ;	//Fault reason 16
  ENB_BEFORE : BOOL ;	//More Faults before
  AU_R : BOOL ;	//Automatic release drive
  LOA : BOOL ;	//Local Mode
  TEXT_F01 { S7_m_c := 'true' }: STRING  [20 ];	//Messagetext Fault_01
  TEXT_F02 { S7_m_c := 'true' }: STRING  [20 ];	//Messagetext Fault_02
  TEXT_F03 { S7_m_c := 'true' }: STRING  [20 ];	//Messagetext Fault_03
  TEXT_F04 { S7_m_c := 'true' }: STRING  [20 ];	//Messagetext Fault_04
  TEXT_F05 { S7_m_c := 'true' }: STRING  [20 ];	//Messagetext Fault_05
  TEXT_F06 { S7_m_c := 'true' }: STRING  [20 ];	//Messagetext Fault_06
  TEXT_F07 { S7_m_c := 'true' }: STRING  [20 ];	//Messagetext Fault_07
  TEXT_F08 { S7_m_c := 'true' }: STRING  [20 ];	//Messagetext Fault_08
  TEXT_F09 { S7_m_c := 'true' }: STRING  [20 ];	//Messagetext Fault_09
  TEXT_F10 { S7_m_c := 'true' }: STRING  [20 ];	//Messagetext Fault_10
  TEXT_F11 { S7_m_c := 'true' }: STRING  [20 ];	//Messagetext Fault_11
  TEXT_F12 { S7_m_c := 'true' }: STRING  [20 ];	//Messagetext Fault_12
  TEXT_F13 { S7_m_c := 'true' }: STRING  [20 ];	//Messagetext Fault_13
  TEXT_F14 { S7_m_c := 'true' }: STRING  [20 ];	//Messagetext Fault_14
  TEXT_F15 { S7_m_c := 'true' }: STRING  [20 ];	//Messagetext Fault_15
  TEXT_F16 { S7_m_c := 'true' }: STRING  [20 ];	//Messagetext Fault_16
END_VAR
VAR_OUTPUT
  ACTUAL_FAULT { S7_m_c := 'true' }: WORD ;	//Actual Fault Code
  LAST_FAULT { S7_m_c := 'true' }: WORD ;	//Last Fault Code
  ENB_DRIVE { S7_m_c := 'true' }: BOOL ;	//Enable to Drive
  ACT_FAULT { S7_m_c := 'true' }: BOOL ;	//Fault is actual
  GONE_FAULT { S7_m_c := 'true' }: BOOL ;	//Fault is gone not acknowledged
  ACK { S7_dynamic := 'true' }: BOOL ;
  Y_LAST_FAULT1 { S7_m_c := 'true' }: BOOL ;	//Not acknowledged Fault 1
  Y_LAST_FAULT2 { S7_m_c := 'true' }: BOOL ;	//Not acknowledged Fault 2
  Y_LAST_FAULT3 { S7_m_c := 'true' }: BOOL ;	//Not acknowledged Fault 3
  Y_LAST_FAULT4 { S7_m_c := 'true' }: BOOL ;	//Not acknowledged Fault 4
  Y_LAST_FAULT5 { S7_m_c := 'true' }: BOOL ;	//Not acknowledged Fault 5
  Y_LAST_FAULT6 { S7_m_c := 'true' }: BOOL ;	//Not acknowledged Fault 6
  Y_LAST_FAULT7 { S7_m_c := 'true' }: BOOL ;	//Not acknowledged Fault 7
  Y_LAST_FAULT8 { S7_m_c := 'true' }: BOOL ;	//Not acknowledged Fault 8
  Y_LAST_FAULT9 { S7_m_c := 'true' }: BOOL ;	//Not acknowledged Fault 9
  Y_LAST_FAULT10 { S7_m_c := 'true' }: BOOL ;	//Not acknowledged Fault 10
  Y_LAST_FAULT11 { S7_m_c := 'true' }: BOOL ;	//Not acknowledged Fault 11
  Y_LAST_FAULT12 { S7_m_c := 'true' }: BOOL ;	//Not acknowledged Fault 12
  Y_LAST_FAULT13 { S7_m_c := 'true' }: BOOL ;	//Not acknowledged Fault 13
  Y_LAST_FAULT14 { S7_m_c := 'true' }: BOOL ;	//Not acknowledged Fault 14
  Y_LAST_FAULT15 { S7_m_c := 'true' }: BOOL ;	//Not acknowledged Fault 15
  Y_LAST_FAULT16 { S7_m_c := 'true' }: BOOL ;	//Not acknowledged Fault 16
END_VAR
VAR_IN_OUT
  ACK_FAULT { S7_m_c := 'true' }: BOOL ;	//Reset faults on this block
  ACK_GEN { S7_m_c := 'true' }: BOOL ;	//Reset all faults in area
  BLOCK { S7_m_c := 'true' }: WORD ;	//Block Fault event
END_VAR
VAR
  AUX_FAULT_NEW : WORD ;
  AUX_FAULT_LAST : WORD ;
  AUX_FAULT_ACT : WORD ;
  AUX_SPARE1 : WORD ;
  AUX_SPARE2 : WORD ;
  AUX_SPARE3 : WORD ;
  AUX_F_01 : BOOL ;
  AUX_F_02 : BOOL ;
  AUX_F_03 : BOOL ;
  AUX_F_04 : BOOL ;
  AUX_F_05 : BOOL ;
  AUX_F_06 : BOOL ;
  AUX_F_07 : BOOL ;
  AUX_F_08 : BOOL ;
  NO_ACT_FAULT : BOOL ;
END_VAR
BEGIN
NETWORK
TITLE =
      L     #AUX_FAULT_NEW;
      T     #AUX_FAULT_ACT;
      L     0;
      T     #AUX_FAULT_NEW;
      AN    #FAULT_01;
      JC    P2;
      L     #AUX_FAULT_NEW;
      L     W#16#1;
      OW;
      T     #AUX_FAULT_NEW;
P2:   AN    #FAULT_02;
      JC    P3;
      L     #AUX_FAULT_NEW;
      L     W#16#2;
      OW;
      T     #AUX_FAULT_NEW;
P3:   AN    #FAULT_03;
      JC    P4;
      L     #AUX_FAULT_NEW;
      L     W#16#4;
      OW;
      T     #AUX_FAULT_NEW;
P4:   AN    #FAULT_04;
      JC    P5;
      L     #AUX_FAULT_NEW;
      L     W#16#6;
      OW;
      T     #AUX_FAULT_NEW;
P5:   AN    #FAULT_05;
      JC    P6;
      L     #AUX_FAULT_NEW;
      L     W#16#10;
      OW;
      T     #AUX_FAULT_NEW;
P6:   AN    #FAULT_06;
      JC    P7;
      L     #AUX_FAULT_NEW;
      L     W#16#20;
      OW;
      T     #AUX_FAULT_NEW;
P7:   AN    #FAULT_07;
      JC    P8;
      L     #AUX_FAULT_NEW;
      L     W#16#40;
      OW;
      T     #AUX_FAULT_NEW;
P8:   AN    #FAULT_08;
      JC    P9;
      L     #AUX_FAULT_NEW;
      L     W#16#80;
      OW;
      T     #AUX_FAULT_NEW;
P9:   AN    #FAULT_09;
      JC    P10;
      L     #AUX_FAULT_NEW;
      L     W#16#100;
      OW;
      T     #AUX_FAULT_NEW;
P10:  AN    #FAULT_10;
      JC    P11;
      L     #AUX_FAULT_NEW;
      L     W#16#200;
      OW;
      T     #AUX_FAULT_NEW;
P11:  AN    #FAULT_11;
      JC    P12;
      L     #AUX_FAULT_NEW;
      L     W#16#400;
      OW;
      T     #AUX_FAULT_NEW;
P12:  AN    #FAULT_12;
      JC    P13;
      L     #AUX_FAULT_NEW;
      L     W#16#600;
      OW;
      T     #AUX_FAULT_NEW;
P13:  AN    #FAULT_13;
      JC    P14;
      L     #AUX_FAULT_NEW;
      L     W#16#1000;
      OW;
      T     #AUX_FAULT_NEW;
P14:  AN    #FAULT_14;
      JC    P15;
      L     #AUX_FAULT_NEW;
      L     W#16#2000;
      OW;
      T     #AUX_FAULT_NEW;
P15:  AN    #FAULT_15;
      JC    P16;
      L     #AUX_FAULT_NEW;
      L     W#16#4000;
      OW;
      T     #AUX_FAULT_NEW;
P16:  AN    #FAULT_16;
      JC    P17;
      L     #AUX_FAULT_NEW;
      L     W#16#8000;
      OW;
      T     #AUX_FAULT_NEW;
P17:  NOP   0;
NETWORK
TITLE =
      L     #AUX_FAULT_NEW;
      L     #BLOCK;
      AW;
      T     #ACTUAL_FAULT;
      L     0;
      <>I;
      =     #ACT_FAULT;
      A     #ENB_BEFORE;
      AN    #ACT_FAULT;
      =     #ENB_DRIVE;
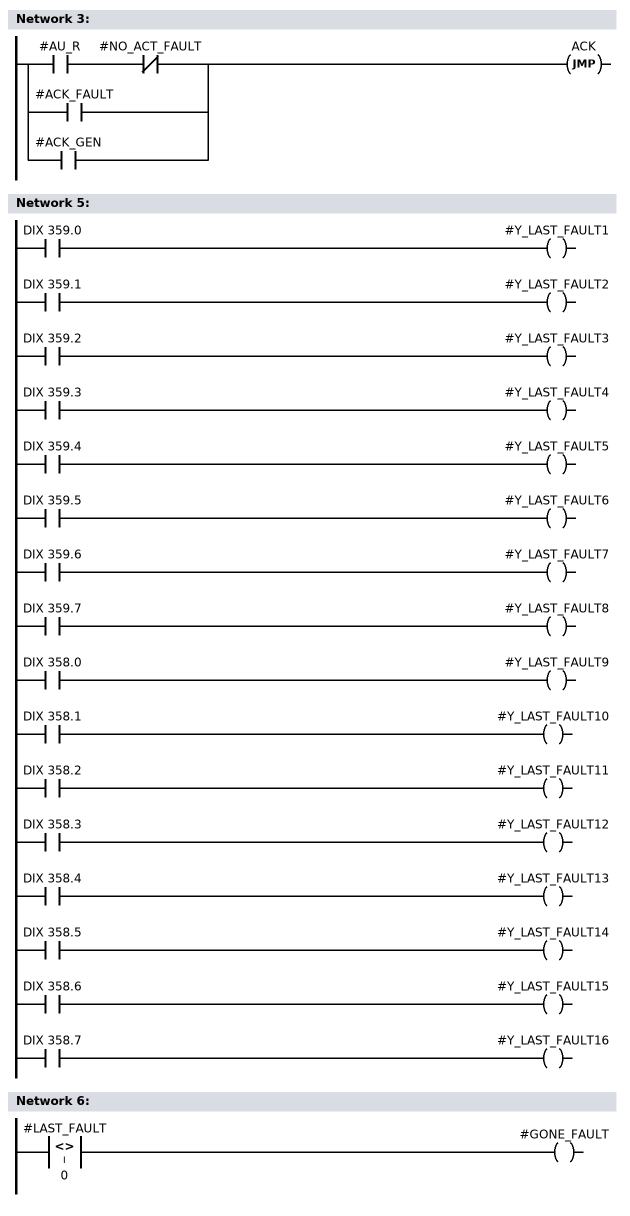
NETWORK
TITLE =
      A     #AU_R;
      AN    #NO_ACT_FAULT;
      O     #ACK_FAULT;
      O     #ACK_GEN;
      JC    ACK;
NETWORK
TITLE =
      O(;
      A     #AU_R;
      AN    #NO_ACT_FAULT;
      );
      O     #ACK_FAULT;
      O     #ACK_GEN;
      JC    ACK;
      L     #ACTUAL_FAULT;
      L     #AUX_FAULT_LAST;
      OW;
      L     #BLOCK;
      AW;
      T     #LAST_FAULT;
      T     #AUX_FAULT_LAST;
      JU    OUT;
ACK:  L     0;
      T     #AUX_FAULT_LAST;
      T     #LAST_FAULT;
OUT:  A     #AU_R;
      JC    AUS;
      JU    AUR;
AUS:  S     #NO_ACT_FAULT;
      JU    AUE;
AUR:  R     #NO_ACT_FAULT;
AUE:  NOP   0;
NETWORK
TITLE =
      A     DIX 359.0;
      =     #Y_LAST_FAULT1;
      A     DIX 359.1;
      =     #Y_LAST_FAULT2;
      A     DIX 359.2;
      =     #Y_LAST_FAULT3;
      A     DIX 359.3;
      =     #Y_LAST_FAULT4;
      A     DIX 359.4;
      =     #Y_LAST_FAULT5;
      A     DIX 359.5;
      =     #Y_LAST_FAULT6;
      A     DIX 359.6;
      =     #Y_LAST_FAULT7;
      A     DIX 359.7;
      =     #Y_LAST_FAULT8;
      A     DIX 358.0;
      =     #Y_LAST_FAULT9;
      A     DIX 358.1;
      =     #Y_LAST_FAULT10;
      A     DIX 358.2;
      =     #Y_LAST_FAULT11;
      A     DIX 358.3;
      =     #Y_LAST_FAULT12;
      A     DIX 358.4;
      =     #Y_LAST_FAULT13;
      A     DIX 358.5;
      =     #Y_LAST_FAULT14;
      A     DIX 358.6;
      =     #Y_LAST_FAULT15;
      A     DIX 358.7;
      =     #Y_LAST_FAULT16;
NETWORK
TITLE =
      L     #LAST_FAULT;
      L     0;
      <>I;
      =     #GONE_FAULT;
NETWORK
TITLE =
      A     #ACK_FAULT;
      O     #ACK_GEN;
      =     #ACK;
      CLR;
      =     #ACK_FAULT;
      =     #ACK_GEN;
END_FUNCTION_BLOCK

FUNCTION_BLOCK "VISU_GEN"	// FB 1067
TITLE = Block to visualize different tags
//==============================
//
//Systemtest   : Pilotierungsstart: 14.09.99
//Abnahme      :
//Änderung #01 :    
//==============================
//KNOW_HOW_PROTECT
//CHANGE #1  : Neue TC-Bibliothek SB1BASE0 und SB1DRIV0 V07.06.00.00; mit PCS7 V6.1 übersetzt    19.12.05
//
AUTHOR : Siemens
FAMILY : Projets
NAME : VISUGEN
VERSION : 0.0
VAR_OUTPUT
  BOOL_1 { S7_m_c := 'true' }: BOOL ;	//BOOL OUTPUT 1
  BOOL_2 { S7_m_c := 'true' }: BOOL ;	//BOOL OUTPUT 2
  BOOL_3 { S7_m_c := 'true' }: BOOL ;	//BOOL OUTPUT 3
  BOOL_4 { S7_m_c := 'true' }: BOOL ;	//BOOL OUTPUT 4
  WORD_1 { S7_m_c := 'true' }: WORD ;	//WORD OUTPUT 1
  WORD_2 { S7_m_c := 'true' }: WORD ;	//WORD OUTPUT 2
  WORD_3 { S7_m_c := 'true' }: WORD ;	//WORD OUTPUT 3
  WORD_4 { S7_m_c := 'true' }: WORD ;	//WORD OUTPUT 4
  DW_1 { S7_m_c := 'true' }: DWORD ;	//DWORD OUTPUT 1
  DW_2 { S7_m_c := 'true' }: DWORD ;	//DWORD OUTPUT 2
  DW_3 { S7_m_c := 'true' }: DWORD ;	//DWORD OUTPUT 3
  DW_4 { S7_m_c := 'true' }: DWORD ;	//DWORD OUTPUT 4
  INT_1 { S7_m_c := 'true' }: INT ;	//INT OUTPUT 1
  INT_2 { S7_m_c := 'true' }: INT ;	//INT OUTPUT 2
  INT_3 { S7_m_c := 'true' }: INT ;	//INT OUTPUT 3
  INT_4 { S7_m_c := 'true' }: INT ;	//INT OUTPUT 4
  DINT_1 { S7_m_c := 'true' }: DINT ;	//DINT OUTPUT 1
  DINT_2 { S7_m_c := 'true' }: DINT ;	//DINT OUTPUT 2
  DINT_3 { S7_m_c := 'true' }: DINT ;	//DINT OUTPUT 3
  DINT_4 { S7_m_c := 'true' }: DINT ;	//DINT OUTPUT 4
  REAL_1 { S7_m_c := 'true' }: REAL ;	//REAL OUTPUT 1
  REAL_2 { S7_m_c := 'true' }: REAL ;	//REAL OUTPUT 2
  REAL_3 { S7_m_c := 'true' }: REAL ;	//REAL OUTPUT 3
  REAL_4 { S7_m_c := 'true' }: REAL ;	//REAL OUTPUT 4
END_VAR
VAR_IN_OUT
  BOOL_1IN { S7_m_c := 'true' }: BOOL ;	//BOOL INPUT 1 FOR INDICATION ON WINCC
  BOOL_2IN { S7_m_c := 'true' }: BOOL ;	//BOOL INPUT 2 FOR INDICATION ON WINCC
  BOOL_3IN { S7_m_c := 'true' }: BOOL ;	//BOOL INPUT 3 FOR INDICATION ON WINCC
  BOOL_4IN { S7_m_c := 'true' }: BOOL ;	//BOOL INPUT 4 FOR INDICATION ON WINCC
  BOOL_IN1 { S7_m_c := 'true' }: BOOL ;	//BOOL INPUT 1 FOR COMMAND FROM WINCC
  BOOL_IN2 { S7_m_c := 'true' }: BOOL ;	//BOOL INPUT 2 FOR COMMAND FROM WINCC
  BOOL_IN3 { S7_m_c := 'true' }: BOOL ;	//BOOL INPUT 3 FOR COMMAND FROM WINCC
  BOOL_IN4 { S7_m_c := 'true' }: BOOL ;	//BOOL INPUT 4 FOR COMMAND FROM WINCC
  WORD_IN1 { S7_m_c := 'true' }: WORD ;	//WORD INPUT 1
  WORD_IN2 { S7_m_c := 'true' }: WORD ;	//WORD INPUT 2
  WORD_IN3 { S7_m_c := 'true' }: WORD ;	//WORD INPUT 3
  WORD_IN4 { S7_m_c := 'true' }: WORD ;	//WORD INPUT 4
  DW_IN1 { S7_m_c := 'true' }: DWORD ;	//DWORD INPUT 1
  DW_IN2 { S7_m_c := 'true' }: DWORD ;	//DWORD INPUT 2
  DW_IN3 { S7_m_c := 'true' }: DWORD ;	//DWORD INPUT 3
  DW_IN4 { S7_m_c := 'true' }: DWORD ;	//DWORD INPUT 4
  INT_IN1 { S7_m_c := 'true' }: INT ;	//INT INPUT 1
  INT_IN2 { S7_m_c := 'true' }: INT ;	//INT INPUT 2
  INT_IN3 { S7_m_c := 'true' }: INT ;	//INT INPUT 3
  INT_IN4 { S7_m_c := 'true' }: INT ;	//INT INPUT 4
  DINT_IN1 { S7_m_c := 'true' }: DINT ;	//DINT INPUT 1
  DINT_IN2 { S7_m_c := 'true' }: DINT ;	//DINT INPUT 2
  DINT_IN3 { S7_m_c := 'true' }: DINT ;	//DINT INPUT 3
  DINT_IN4 { S7_m_c := 'true' }: DINT ;	//DINT INPUT 4
  REAL_IN1 { S7_m_c := 'true' }: REAL ;	//REAL INPUT 1
  REAL_IN2 { S7_m_c := 'true' }: REAL ;	//REAL INPUT 2
  REAL_IN3 { S7_m_c := 'true' }: REAL ;	//REAL INPUT 3
  REAL_IN4 { S7_m_c := 'true' }: REAL ;	//REAL INPUT 4
END_VAR
VAR
  BOOL_AUX1 : BOOL ;	//AUXILIARY BOOL 1
  BOOL_AUX2 : BOOL ;	//AUXILIARY BOOL 2
  BOOL_AUX3 : BOOL ;	//AUXILIARY BOOL 3
  BOOL_AUX4 : BOOL ;	//AUXILIARY BOOL 4
END_VAR
BEGIN
NETWORK
TITLE = SCL network
//compiled by SCL compiler version:  SCL K4.0.2 (K4.0.9.5)
      SET;
      SAVE;
      =     L 0.1;
      A     #BOOL_IN1;
      =     #BOOL_AUX1;
      A     #BOOL_IN2;
      =     #BOOL_AUX2;
      A     #BOOL_IN3;
      =     #BOOL_AUX3;
      A     #BOOL_IN4;
      =     #BOOL_AUX4;
      A     #BOOL_AUX1;
      =     #BOOL_1;
      A     #BOOL_AUX2;
      =     #BOOL_2;
      A     #BOOL_AUX3;
      =     #BOOL_3;
      A     #BOOL_AUX4;
      =     #BOOL_4;
      A     #BOOL_AUX1;
      JCN   A7d0;
      CLR;
      =     #BOOL_IN1;
A7d0: CLR;
      A     #BOOL_AUX2;
      JCN   A7d1;
      CLR;
      =     #BOOL_IN2;
A7d1: CLR;
      A     #BOOL_AUX3;
      JCN   A7d2;
      CLR;
      =     #BOOL_IN3;
A7d2: CLR;
      A     #BOOL_AUX4;
      JCN   A7d3;
      CLR;
      =     #BOOL_IN4;
A7d3: L     #WORD_IN1;
      T     #WORD_1;
      L     #WORD_IN2;
      T     #WORD_2;
      L     #WORD_IN3;
      T     #WORD_3;
      L     #WORD_IN4;
      T     #WORD_4;
      L     #DW_IN1;
      T     #DW_1;
      L     #DW_IN2;
      T     #DW_2;
      L     #DW_IN3;
      T     #DW_3;
      L     #DW_IN4;
      T     #DW_4;
      L     #INT_IN1;
      T     #INT_1;
      L     #INT_IN2;
      T     #INT_2;
      L     #INT_IN3;
      T     #INT_3;
      L     #INT_IN4;
      T     #INT_4;
      L     #DINT_IN1;
      T     #DINT_1;
      L     #DINT_IN2;
      T     #DINT_2;
      L     #DINT_IN3;
      T     #DINT_3;
      L     #DINT_IN4;
      T     #DINT_4;
      L     #REAL_IN1;
      T     #REAL_1;
      L     #REAL_IN2;
      T     #REAL_2;
      L     #REAL_IN3;
      T     #REAL_3;
      L     #REAL_IN4;
      T     #REAL_4;
      CLR;
      A     L 0.1;
      SAVE;
      BE;
END_FUNCTION_BLOCK

FUNCTION_BLOCK "N_AnMeas"	// FB 1435
VERSION : 0.1
VAR_INPUT
  CFG { S7_dynamic := 'true' }: BOOL ;	//0 - input XE used if 1 - PV - used, no scaling inside block
  PV { S7_dynamic := 'true' }: REAL ;
  XE { S7_dynamic := 'true' }: WORD ;	//Input word
  MR_FIN { S7_dynamic := 'true' }: REAL ;	//Measuring range final
  MR_INI { S7_dynamic := 'true' }: REAL ;	//Measuring range initial
  VA_UP { S7_dynamic := 'true' }: INT ;	//Digits value abnormal upper
  VA_LOW { S7_dynamic := 'true' }: INT ;	//Digits value abnormal lower
  CODE { S7_string_0 := '0..+/4-20mA/1-5V'; S7_string_1 := 'Range - .... +' }: BOOL ;	//Type of input card
  EN_LIM { S7_string_0 := 'Y not limited'; S7_string_1 := 'Y limited' }: BOOL ;	//Limit output to measuring range
  HH_LIM { S7_dynamic := 'true'; S7_m_c := 'true' }: REAL ;
  H_LIM { S7_m_c := 'true'; S7_dynamic := 'true' }: REAL ;
  L_LIM { S7_dynamic := 'true'; S7_m_c := 'true' }: REAL ;
  LL_LIM { S7_dynamic := 'true'; S7_m_c := 'true' }: REAL ;
  MONDELAY { S7_dynamic := 'true' }: TIME ;
  HYST { S7_dynamic := 'true'; S7_m_c := 'true' }: REAL ;
  SIM { S7_dynamic := 'true' }: BOOL ;
  SIMVAL { S7_dynamic := 'true' }: REAL ;	//Simulation Value
  MASK { S7_dynamic := 'true'; S7_m_c := 'true' }: WORD ;
  EVID { S7_a_type := 'alarm_8p'; S7_server := 'alarm_archiv' }: DWORD ;
  Ack { S7_dynamic := 'true' }: BOOL ;
END_VAR
VAR_OUTPUT
  HH_ALARM : BOOL ;
  H_ALARM : BOOL ;
  L_ALARM : BOOL ;
  LL_ALARM : BOOL ;
  DEVERR { S7_dynamic := 'true' }: BOOL ;
  MV { S7_dynamic := 'true'; S7_m_c := 'true'; S7_unit := '' }: REAL ;
  STATUS { S7_m_c := 'true'; S7_dynamic := 'true' }: INT ;
END_VAR
VAR
  HHTON : SFB 4;
  HTON : SFB 4;
  LTON : SFB 4;
  LLTON : SFB 4;
  HMIStatus : FB 982;
  Alarms : SFB 35;
  Stat : STRUCT
   HH_Alarm : BOOL ;
   H_Alarm : BOOL ;
   L_Alarm : BOOL ;
   LL_Alarm : BOOL ;
   Dev_Err : BOOL ;
   Byp_Act : BOOL ;
   Spare : BOOL ;
   Spare_1 : BOOL ;
   Spare_2 : BOOL ;
   Spare_3 : BOOL ;
   Spare_4 : BOOL ;
   Spare_5 : BOOL ;
   Spare_6 : BOOL ;
   Spare_7 : BOOL ;
   Spare_8 : BOOL ;
   Spare_9 : BOOL ;
  END_STRUCT ;
  Meas : REAL ;
  temp_bool : BOOL ;
  HH_Alarm_Int : BOOL ;
  H_Alarm_Int : BOOL ;
  L_Alarm_Int : BOOL ;
  LL_Alarm_Int : BOOL ;
END_VAR
VAR_TEMP
  Log_0 : BOOL ;
  Log_1 : BOOL ;
  Temp_Real : REAL ;
  HHNODELAY : BOOL ;
  HNODELAY : BOOL ;
  LNODELAY : BOOL ;
  LLNODELAY : BOOL ;
  ZeroDelay : BOOL ;
  HH_Mask : BOOL ;
  H_Mask : BOOL ;
  L_Mask : BOOL ;
  LL_Mask : BOOL ;
  DevErr_Mask : BOOL ;
  Dummy_Int : INT ;
END_VAR
BEGIN
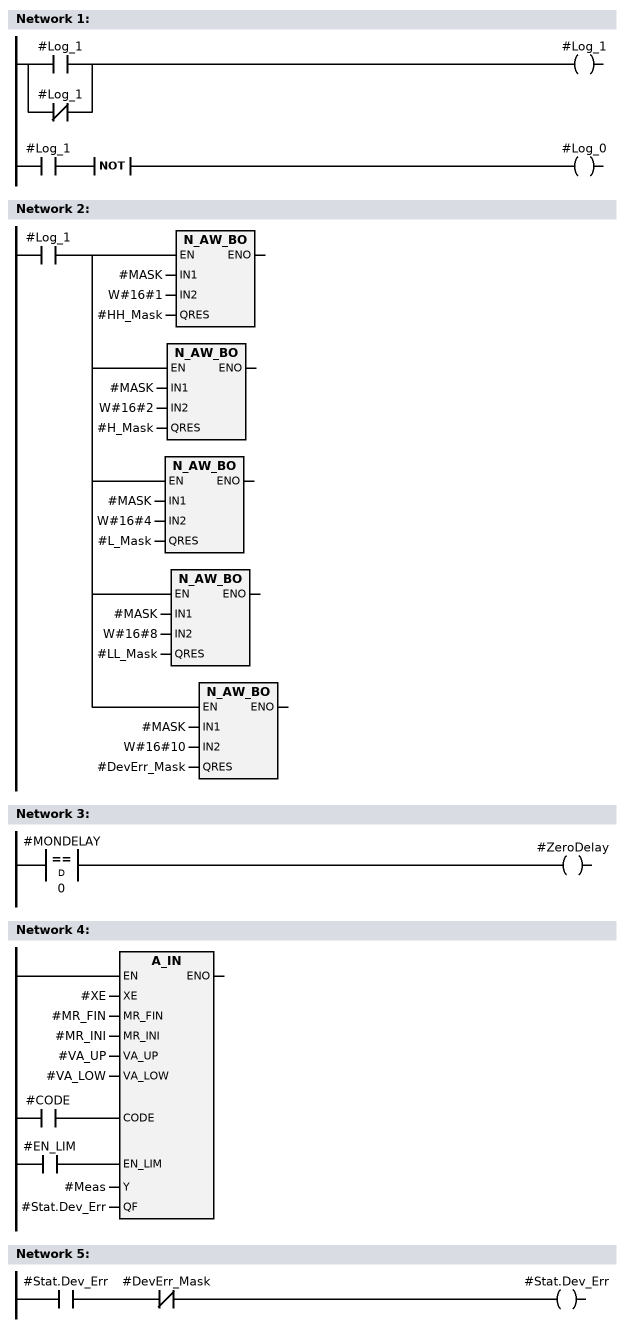
NETWORK
TITLE =
      A(;
      O     #Log_1;
      ON    #Log_1;
      );
      =     #Log_1;
      A     #Log_1;
      NOT;
      =     #Log_0;
NETWORK
TITLE =
      A     #Log_1;
      =     L 10.0;
      A     L 10.0;
      JNB   _001;
      CALL  "N_AW_BO" (
           IN1                      := #MASK,
           IN2                      := W#16#1,
           QRES                     := #HH_Mask);
_001: NOP   0;
      A     L 10.0;
      JNB   _002;
      CALL  "N_AW_BO" (
           IN1                      := #MASK,
           IN2                      := W#16#2,
           QRES                     := #H_Mask);
_002: NOP   0;
      A     L 10.0;
      JNB   _003;
      CALL  "N_AW_BO" (
           IN1                      := #MASK,
           IN2                      := W#16#4,
           QRES                     := #L_Mask);
_003: NOP   0;
      A     L 10.0;
      JNB   _007;
      CALL  "N_AW_BO" (
           IN1                      := #MASK,
           IN2                      := W#16#8,
           QRES                     := #LL_Mask);
_007: NOP   0;
      A     L 10.0;
      JNB   _010;
      CALL  "N_AW_BO" (
           IN1                      := #MASK,
           IN2                      := W#16#10,
           QRES                     := #DevErr_Mask);
_010: NOP   0;
NETWORK
TITLE =
      L     #MONDELAY;
      L     0;
      ==D;
      =     #ZeroDelay;
NETWORK
TITLE =
      A     #CODE;
      =     L 10.0;
      BLD   103;
      A     #EN_LIM;
      =     L 10.1;
      BLD   103;
      CALL  "A_IN" (
           XE                       := #XE,
           MR_FIN                   := #MR_FIN,
           MR_INI                   := #MR_INI,
           VA_UP                    := #VA_UP,
           VA_LOW                   := #VA_LOW,
           CODE                     := L 10.0,
           EN_LIM                   := L 10.1,
           Y                        := #Meas,
           QF                       := #Stat.Dev_Err);
      NOP   0;
NETWORK
TITLE =
      A     #Stat.Dev_Err;
      AN    #DevErr_Mask;
      =     #Stat.Dev_Err;
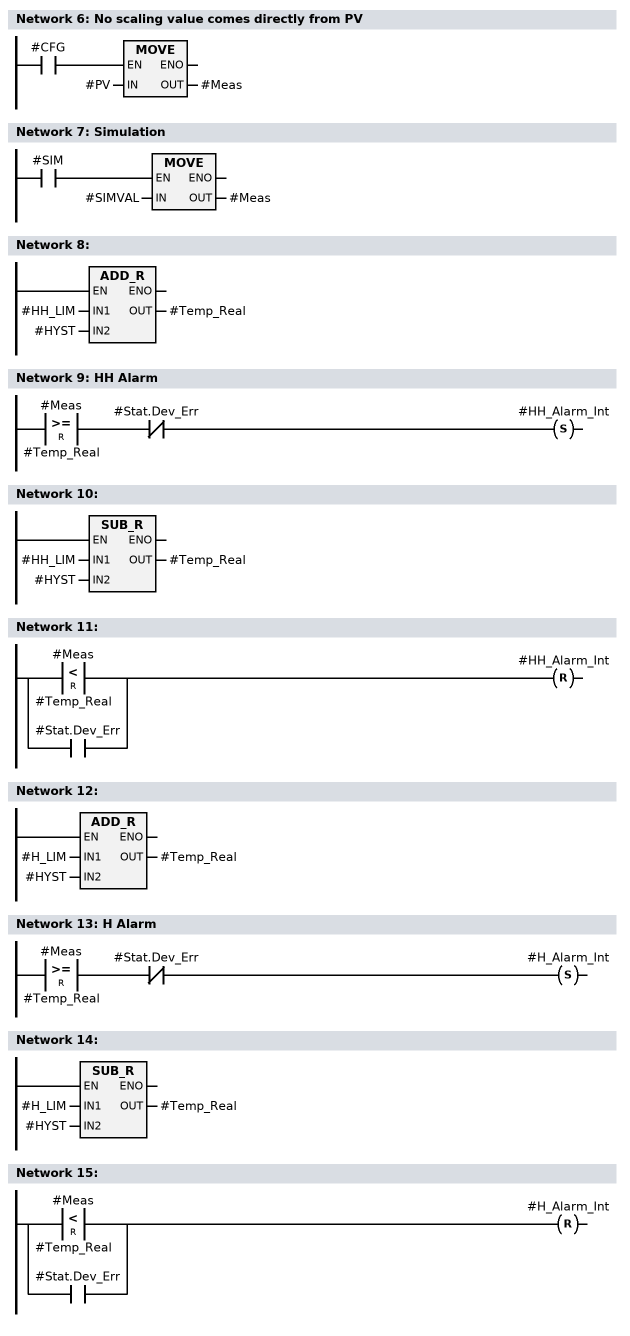
NETWORK
TITLE = No scaling value comes directly from PV
      A     #CFG;
      JNB   _011;
      L     #PV;
      T     #Meas;
_011: NOP   0;
NETWORK
TITLE = Simulation
      A     #SIM;
      JNB   _012;
      L     #SIMVAL;
      T     #Meas;
_012: NOP   0;
NETWORK
TITLE =
      L     #HH_LIM;
      L     #HYST;
      +R;
      T     #Temp_Real;
      NOP   0;
NETWORK
TITLE = HH Alarm
      A(;
      L     #Meas;
      L     #Temp_Real;
      >=R;
      );
      AN    #Stat.Dev_Err;
      S     #HH_Alarm_Int;
NETWORK
TITLE =
      L     #HH_LIM;
      L     #HYST;
      -R;
      T     #Temp_Real;
      NOP   0;
NETWORK
TITLE =
      O(;
      L     #Meas;
      L     #Temp_Real;
      <R;
      );
      O     #Stat.Dev_Err;
      R     #HH_Alarm_Int;
NETWORK
TITLE =
      L     #H_LIM;
      L     #HYST;
      +R;
      T     #Temp_Real;
      NOP   0;
NETWORK
TITLE = H Alarm
      A(;
      L     #Meas;
      L     #Temp_Real;
      >=R;
      );
      AN    #Stat.Dev_Err;
      S     #H_Alarm_Int;
NETWORK
TITLE =
      L     #H_LIM;
      L     #HYST;
      -R;
      T     #Temp_Real;
      NOP   0;
NETWORK
TITLE =
      O(;
      L     #Meas;
      L     #Temp_Real;
      <R;
      );
      O     #Stat.Dev_Err;
      R     #H_Alarm_Int;
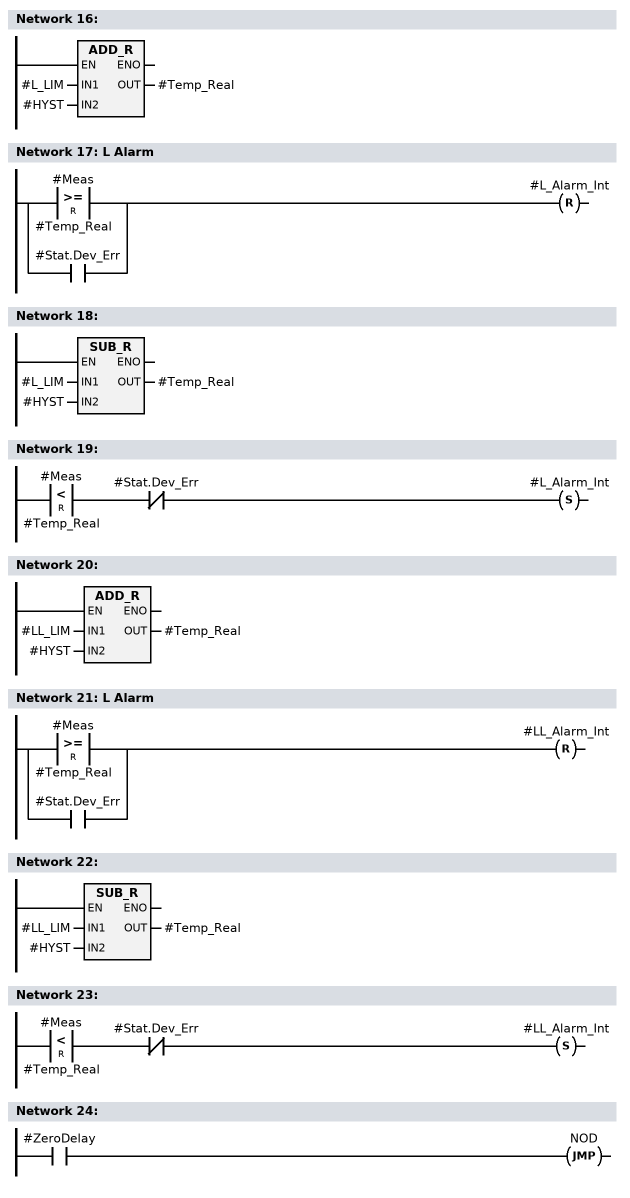
NETWORK
TITLE =
      L     #L_LIM;
      L     #HYST;
      +R;
      T     #Temp_Real;
      NOP   0;
NETWORK
TITLE = L Alarm
      O(;
      L     #Meas;
      L     #Temp_Real;
      >=R;
      );
      O     #Stat.Dev_Err;
      R     #L_Alarm_Int;
NETWORK
TITLE =
      L     #L_LIM;
      L     #HYST;
      -R;
      T     #Temp_Real;
      NOP   0;
NETWORK
TITLE =
      A(;
      L     #Meas;
      L     #Temp_Real;
      <R;
      );
      AN    #Stat.Dev_Err;
      S     #L_Alarm_Int;
NETWORK
TITLE =
      L     #LL_LIM;
      L     #HYST;
      +R;
      T     #Temp_Real;
      NOP   0;
NETWORK
TITLE = L Alarm
      O(;
      L     #Meas;
      L     #Temp_Real;
      >=R;
      );
      O     #Stat.Dev_Err;
      R     #LL_Alarm_Int;
NETWORK
TITLE =
      L     #LL_LIM;
      L     #HYST;
      -R;
      T     #Temp_Real;
      NOP   0;
NETWORK
TITLE =
      A(;
      L     #Meas;
      L     #Temp_Real;
      <R;
      );
      AN    #Stat.Dev_Err;
      S     #LL_Alarm_Int;
NETWORK
TITLE =
      A     #ZeroDelay;
      JC    NOD;
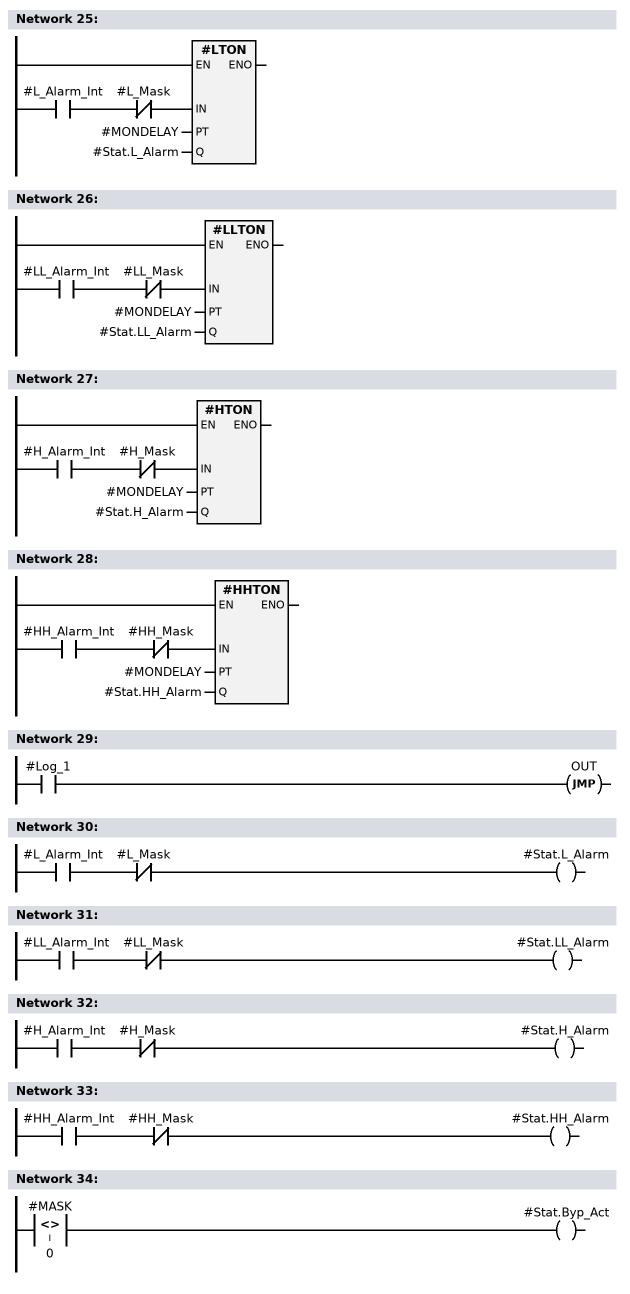
NETWORK
TITLE =
      A     #L_Alarm_Int;
      AN    #L_Mask;
      =     L 10.0;
      BLD   103;
      CALL  #LTON (
           IN                       := L 10.0,
           PT                       := #MONDELAY,
           Q                        := #Stat.L_Alarm);
      NOP   0;
NETWORK
TITLE =
      A     #LL_Alarm_Int;
      AN    #LL_Mask;
      =     L 10.0;
      BLD   103;
      CALL  #LLTON (
           IN                       := L 10.0,
           PT                       := #MONDELAY,
           Q                        := #Stat.LL_Alarm);
      NOP   0;
NETWORK
TITLE =
      A     #H_Alarm_Int;
      AN    #H_Mask;
      =     L 10.0;
      BLD   103;
      CALL  #HTON (
           IN                       := L 10.0,
           PT                       := #MONDELAY,
           Q                        := #Stat.H_Alarm);
      NOP   0;
NETWORK
TITLE =
      A     #HH_Alarm_Int;
      AN    #HH_Mask;
      =     L 10.0;
      BLD   103;
      CALL  #HHTON (
           IN                       := L 10.0,
           PT                       := #MONDELAY,
           Q                        := #Stat.HH_Alarm);
      NOP   0;
NETWORK
TITLE =
      A     #Log_1;
      JC    OUT;
NETWORK
TITLE =
NOD:  A     #L_Alarm_Int;
      AN    #L_Mask;
      =     #Stat.L_Alarm;
NETWORK
TITLE =
      A     #LL_Alarm_Int;
      AN    #LL_Mask;
      =     #Stat.LL_Alarm;
NETWORK
TITLE =
      A     #H_Alarm_Int;
      AN    #H_Mask;
      =     #Stat.H_Alarm;
NETWORK
TITLE =
      A     #HH_Alarm_Int;
      AN    #HH_Mask;
      =     #Stat.HH_Alarm;
NETWORK
TITLE =
OUT:  L     #MASK;
      L     0;
      <>I;
      =     #Stat.Byp_Act;
NETWORK
TITLE = Alarms
      A     #Stat.HH_Alarm;
      =     L 10.1;
      BLD   103;
      A     #Stat.H_Alarm;
      =     L 10.2;
      BLD   103;
      A     #Stat.L_Alarm;
      =     L 10.3;
      BLD   103;
      A     #Stat.LL_Alarm;
      =     L 10.4;
      BLD   103;
      A     #Stat.Dev_Err;
      =     L 10.5;
      BLD   103;
      BLD   16;
      =     L 18.0;
      L     DINO;
      T     LW 16;
      CDB;
      OPN   DI [LW 16];
      TAR2  LD 12;
      A     L 10.1;
      =     #Alarms.SIG_1;
      A     L 10.2;
      =     #Alarms.SIG_2;
      A     L 10.3;
      =     #Alarms.SIG_3;
      A     L 10.4;
      =     #Alarms.SIG_4;
      A     L 10.5;
      =     #Alarms.SIG_5;
      L     -4370;
      T     #Alarms.ID;
      L     DBD [AR2,P#54.0];
      T     #Alarms.EV_ID;
      L     W#16#1008;
      T     DIW [AR2,P#178.0];
      L     1;
      T     DIW [AR2,P#180.0];
      L     DBNO;
      T     DIW [AR2,P#182.0];
      +AR2  P#22.0;
      TAR2;
      LAR2  LD 12;
      T     DID [AR2,P#184.0];
      L     W#16#1008;
      T     DIW [AR2,P#188.0];
      L     1;
      T     DIW [AR2,P#190.0];
      L     DBNO;
      T     DIW [AR2,P#192.0];
      +AR2  P#26.0;
      TAR2;
      LAR2  LD 12;
      T     DID [AR2,P#194.0];
      L     W#16#1008;
      T     DIW [AR2,P#198.0];
      L     1;
      T     DIW [AR2,P#200.0];
      L     DBNO;
      T     DIW [AR2,P#202.0];
      +AR2  P#30.0;
      TAR2;
      LAR2  LD 12;
      T     DID [AR2,P#204.0];
      L     W#16#1008;
      T     DIW [AR2,P#208.0];
      L     1;
      T     DIW [AR2,P#210.0];
      L     DBNO;
      T     DIW [AR2,P#212.0];
      +AR2  P#34.0;
      TAR2;
      LAR2  LD 12;
      T     DID [AR2,P#214.0];
      +AR2  P#162.0;
      UC    "ALARM_8P";
      LAR2  LD 12;
      CDB;
      BLD   17;
      NOP   0;
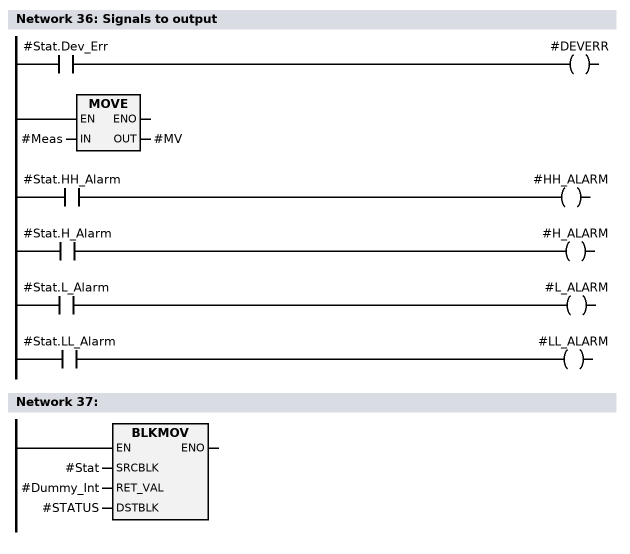
NETWORK
TITLE = Signals to output
      A     #Stat.Dev_Err;
      =     #DEVERR;
      L     #Meas;
      T     #MV;
      A     #Stat.HH_Alarm;
      =     #HH_ALARM;
      A     #Stat.H_Alarm;
      =     #H_ALARM;
      A     #Stat.L_Alarm;
      =     #L_ALARM;
      A     #Stat.LL_Alarm;
      =     #LL_ALARM;
NETWORK
TITLE =
      CALL  "BLKMOV" (
           SRCBLK                   := #Stat,
           RET_VAL                  := #Dummy_Int,
           DSTBLK                   := #STATUS);
      NOP   0;
END_FUNCTION_BLOCK

FUNCTION_BLOCK "N_SPMANIP"	// FB 1467
VERSION : 0.1
VAR_INPUT
  CFG : BOOL ;	//0 INC/DEC by time 1 - INC/DEC by value
  NSC : BOOL ;
  OPT : BOOL ;
  H_LIM : REAL ;
  L_LIM : REAL ;
  RAMP_TIME : TIME ;	//Ramp up time [s]
  DVAL : REAL ;
  CU : BOOL ;
  CD : BOOL ;
  S_SP : REAL ;
END_VAR
VAR_OUTPUT
  QOPT : BOOL ;
  O_SP : REAL ;
  QSP : REAL ;
END_VAR
VAR_IN_OUT
  XSP { S7_m_c := 'true' }: REAL ;
END_VAR
VAR
  New_PV : BOOL ;
  OldTime : TIME ;
  NewTime : TIME ;
  Delta_t : REAL ;
  Ramp_Up_Time : REAL ;
  Ramp_Down_Time : REAL ;
  Current_Val : REAL ;
  Time_to : REAL ;
  Old_PV : REAL ;
  Delta_Val : REAL ;
  PV_Int : REAL ;
  Delta_Up : REAL ;
  Delta_Down : REAL ;
  PV_ABS : REAL ;
  Cur_Val_ABS : REAL ;
  CU_Pulse : BOOL ;
  CD_Pulse : BOOL ;
  Pulse_NSC : BOOL ;
  Pulse_OPT : BOOL ;
END_VAR
VAR_TEMP
  temp_real : REAL ;
  delat_val : BOOL ;
  TEMP2 : BOOL ;
  VAL_RAMP : BOOL ;
  TIME_RAMP : BOOL ;
END_VAR
BEGIN
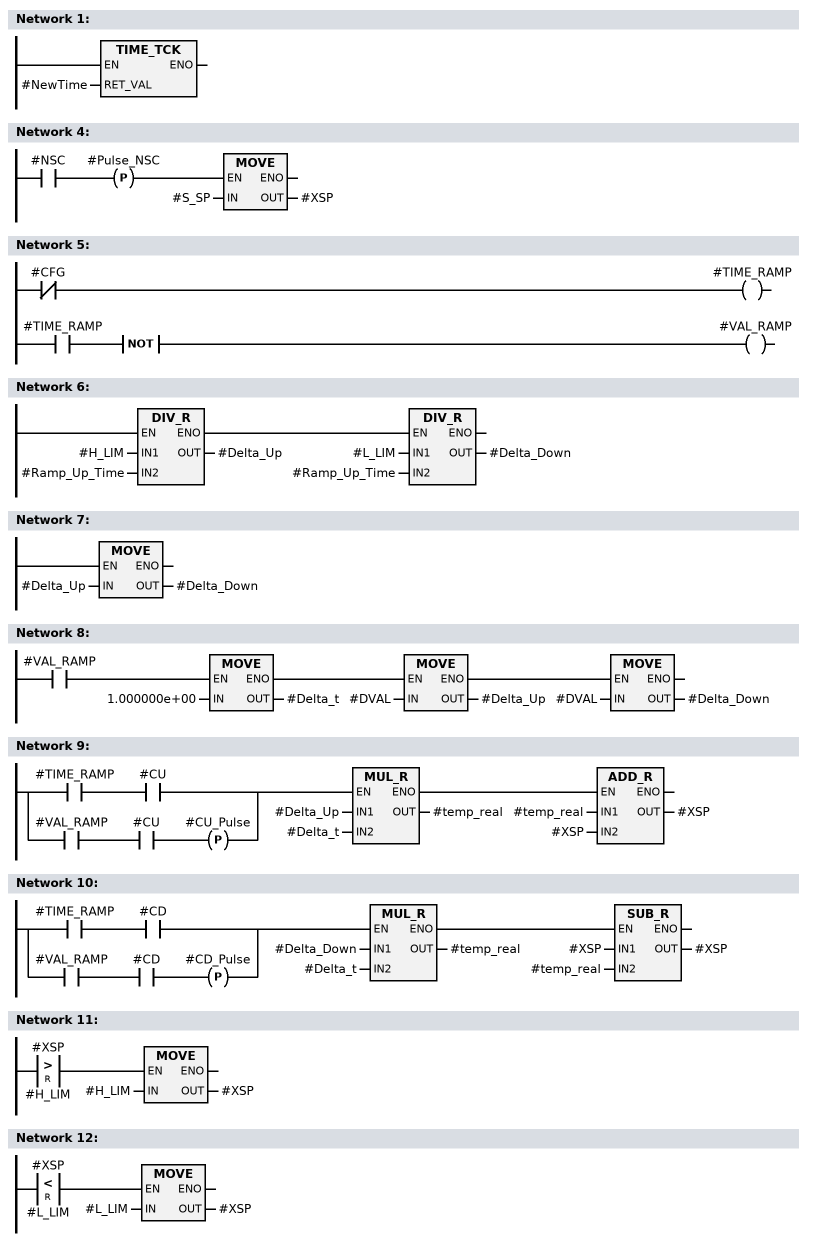
NETWORK
TITLE =
      CALL  "TIME_TCK" (
           RET_VAL                  := #NewTime);
      NOP   0;
NETWORK
TITLE =
      L     #NewTime;
      L     #OldTime;
      -D;
      AD    DW#16#7FFFFFFF;
      DTR;
      L     1.000000e+03;
      /R;
      T     #Delta_t;
      L     #NewTime;
      T     #OldTime;
NETWORK
TITLE =
      L     #RAMP_TIME;
      DTR;
      L     1.000000e+03;
      /R;
      T     #Ramp_Up_Time;
NETWORK
TITLE =
      A     #NSC;
      FP    #Pulse_NSC;
      JNB   _005;
      L     #S_SP;
      T     #XSP;
_005: NOP   0;
NETWORK
TITLE =
//     L     #PV_Int
//      ABS   
//      T     #temp_real
//      L     #Current_Val
//      ABS   
//      L     #temp_real
//      ==R   
//      JCN   M001
//      L     0.000000e+000
//      T     #Delta_t
//M001: NOP   0
      AN    #CFG;
      =     #TIME_RAMP;
      A     #TIME_RAMP;
      NOT;
      =     #VAL_RAMP;
NETWORK
TITLE =
      A(;
      L     #H_LIM;
      L     #Ramp_Up_Time;
      /R;
      T     #Delta_Up;
      AN    OV;
      SAVE;
      CLR;
      A     BR;
      );
      JNB   _006;
      L     #L_LIM;
      L     #Ramp_Up_Time;
      /R;
      T     #Delta_Down;
_006: NOP   0;
NETWORK
TITLE =
      L     #Delta_Up;
      T     #Delta_Down;
      NOP   0;
NETWORK
TITLE =
      A(;
      A(;
      A     #VAL_RAMP;
      JNB   _007;
      L     1.000000e+00;
      T     #Delta_t;
      SET;
      SAVE;
      CLR;
_007: A     BR;
      );
      JNB   _00f;
      L     #DVAL;
      T     #Delta_Up;
      SET;
      SAVE;
      CLR;
_00f: A     BR;
      );
      JNB   _013;
      L     #DVAL;
      T     #Delta_Down;
_013: NOP   0;
NETWORK
TITLE =
      A(;
      A(;
      A     #TIME_RAMP;
      A     #CU;
      O(;
      A     #VAL_RAMP;
      A(;
      A     #CU;
      FP    #CU_Pulse;
      );
      );
      );
      JNB   _02c;
      L     #Delta_Up;
      L     #Delta_t;
      *R;
      T     #temp_real;
      AN    OV;
      SAVE;
      CLR;
_02c: A     BR;
      );
      JNB   _02d;
      L     #temp_real;
      L     #XSP;
      +R;
      T     #XSP;
_02d: NOP   0;
NETWORK
TITLE =
      A(;
      A(;
      A     #TIME_RAMP;
      A     #CD;
      O(;
      A     #VAL_RAMP;
      A(;
      A     #CD;
      FP    #CD_Pulse;
      );
      );
      );
      JNB   _02e;
      L     #Delta_Down;
      L     #Delta_t;
      *R;
      T     #temp_real;
      AN    OV;
      SAVE;
      CLR;
_02e: A     BR;
      );
      JNB   _02f;
      L     #XSP;
      L     #temp_real;
      -R;
      T     #XSP;
_02f: NOP   0;
NETWORK
TITLE =
      A(;
      L     #XSP;
      L     #H_LIM;
      >R;
      );
      JNB   _037;
      L     #H_LIM;
      T     #XSP;
_037: NOP   0;
NETWORK
TITLE =
      A(;
      L     #XSP;
      L     #L_LIM;
      <R;
      );
      JNB   _03b;
      L     #L_LIM;
      T     #XSP;
_03b: NOP   0;
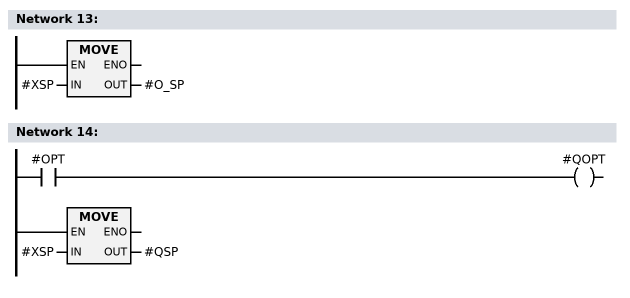
NETWORK
TITLE =
      L     #XSP;
      T     #O_SP;
      NOP   0;
NETWORK
TITLE =
      A     #OPT;
      =     #QOPT;
      L     #XSP;
      T     #QSP;
END_FUNCTION_BLOCK

FUNCTION_BLOCK "N_TON"	// FB 1482
VERSION : 0.1
VAR_INPUT
  IN : BOOL ;
  PT : TIME ;
END_VAR
VAR_OUTPUT
  QIN : BOOL ;
  ET : TIME ;
END_VAR
VAR
  TMR : SFB 4;
END_VAR
VAR_TEMP
  Zero_Delay : BOOL ;
  Tmp_Time : TIME ;
  res : BOOL ;
END_VAR
BEGIN
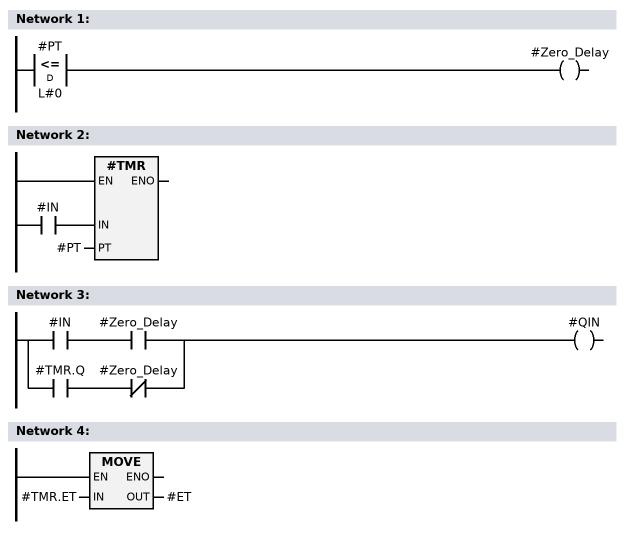
NETWORK
TITLE =
      L     #PT;
      L     L#0;
      <=D;
      =     #Zero_Delay;
NETWORK
TITLE =
      A     #IN;
      =     L 7.0;
      BLD   103;
      CALL  #TMR (
           IN                       := L 7.0,
           PT                       := #PT);
      NOP   0;
NETWORK
TITLE =
      A     #IN;
      A     #Zero_Delay;
      O;
      A     #TMR.Q;
      AN    #Zero_Delay;
      =     #QIN;
NETWORK
TITLE =
      L     #TMR.ET;
      T     #ET;
END_FUNCTION_BLOCK

FUNCTION_BLOCK "N_TOF"	// FB 1483
VERSION : 0.1
VAR_INPUT
  IN : BOOL ;
  PT : TIME ;
END_VAR
VAR_OUTPUT
  QIN : BOOL ;
  ET : TIME ;
END_VAR
VAR
  TMR : SFB 5;
END_VAR
VAR_TEMP
  Zero_Delay : BOOL ;
  Tmp_Time : TIME ;
  res : BOOL ;
END_VAR
BEGIN
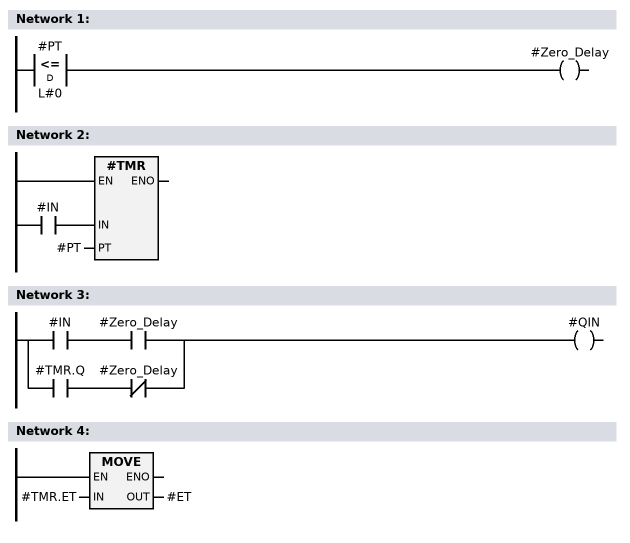
NETWORK
TITLE =
      L     #PT;
      L     L#0;
      <=D;
      =     #Zero_Delay;
NETWORK
TITLE =
      A     #IN;
      =     L 7.0;
      BLD   103;
      CALL  #TMR (
           IN                       := L 7.0,
           PT                       := #PT);
      NOP   0;
NETWORK
TITLE =
      A     #IN;
      A     #Zero_Delay;
      O;
      A     #TMR.Q;
      AN    #Zero_Delay;
      =     #QIN;
NETWORK
TITLE =
      L     #TMR.ET;
      T     #ET;
END_FUNCTION_BLOCK

FUNCTION_BLOCK "CUT_SHER"	// FB 3333
VERSION : 0.1
VAR_INPUT
  CUT_HMD : BOOL ;
  SPID_HMD : REAL ;
  LOC_HMD_SHER : REAL ;
  REF_CUT_HEAD : REAL ;
  CUT : BOOL ;
  HW_TIM_SH : REAL ;
  REF_CUT_TAIL : REAL ;
  ENB_HEAD : BOOL ;
  ENB_TAIL : BOOL ;
END_VAR
VAR_OUTPUT
  CUT_HEAD : BOOL ;
  CUT_TEAL : BOOL ;
  TIM_HEAD_ALL : REAL ;
  TIM_TEAL_ALL : REAL ;
END_VAR
VAR
  TIM_HEAD_1 : REAL ;
  TIM_HEAD_2 : REAL ;
  TIM_HEAD_3 : REAL ;
  CUT_HMD_PULS : BOOL ;
  PULS_1_0 : BOOL ;
  PULS_1_3 : BOOL ;
  PULS_1_2 : BOOL ;
  PULS_1_1 : BOOL ;
  PULS_1_4 : BOOL ;
  TIM_TEAL_1 : REAL ;
  TIM_TEAL_2 : REAL ;
  TIM_TEAL_3 : REAL ;
  HEAD_RELIZ : BOOL ;
  TAIL_RELIZ : BOOL ;
END_VAR
BEGIN
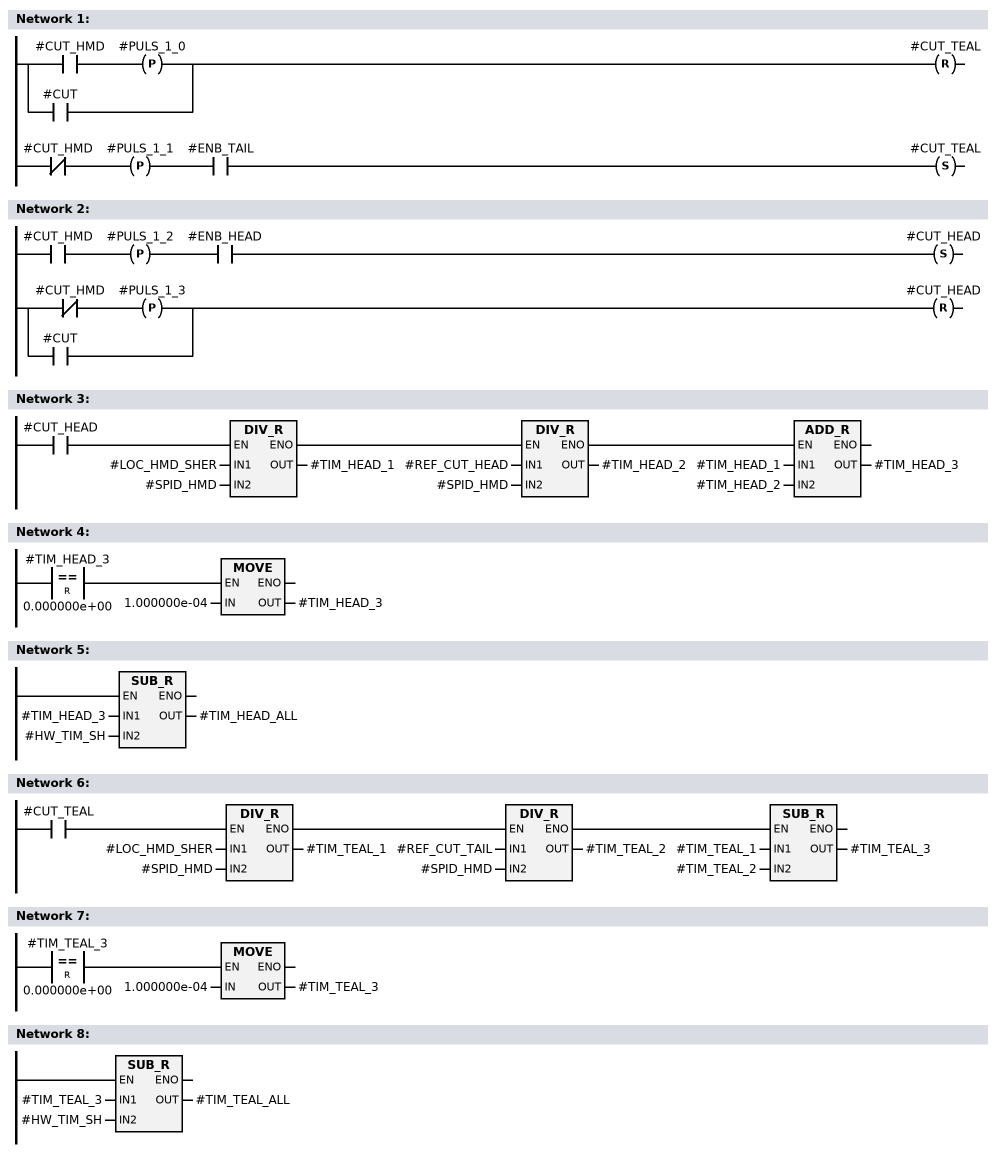
NETWORK
TITLE =
      A(;
      A     #CUT_HMD;
      FP    #PULS_1_0;
      O     #CUT;
      );
      R     #CUT_TEAL;
      AN    #CUT_HMD;
      FP    #PULS_1_1;
      A     #ENB_TAIL;
      S     #CUT_TEAL;
      NOP   0;
NETWORK
TITLE =
      A     #CUT_HMD;
      FP    #PULS_1_2;
      A     #ENB_HEAD;
      S     #CUT_HEAD;
      A(;
      AN    #CUT_HMD;
      FP    #PULS_1_3;
      O     #CUT;
      );
      R     #CUT_HEAD;
      NOP   0;
NETWORK
TITLE =
      A(;
      A(;
      A     #CUT_HEAD;
      JNB   _001;
      L     #LOC_HMD_SHER;
      L     #SPID_HMD;
      /R;
      T     #TIM_HEAD_1;
      AN    OV;
      SAVE;
      CLR;
_001: A     BR;
      );
      JNB   _002;
      L     #REF_CUT_HEAD;
      L     #SPID_HMD;
      /R;
      T     #TIM_HEAD_2;
      AN    OV;
      SAVE;
      CLR;
_002: A     BR;
      );
      JNB   _003;
      L     #TIM_HEAD_1;
      L     #TIM_HEAD_2;
      +R;
      T     #TIM_HEAD_3;
_003: NOP   0;
NETWORK
TITLE =
      A(;
      L     #TIM_HEAD_3;
      L     0.000000e+00;
      ==R;
      );
      JNB   _004;
      L     1.000000e-04;
      T     #TIM_HEAD_3;
_004: NOP   0;
NETWORK
TITLE =
      L     #TIM_HEAD_3;
      L     #HW_TIM_SH;
      -R;
      T     #TIM_HEAD_ALL;
      NOP   0;
NETWORK
TITLE =
      A(;
      A(;
      A     #CUT_TEAL;
      JNB   _005;
      L     #LOC_HMD_SHER;
      L     #SPID_HMD;
      /R;
      T     #TIM_TEAL_1;
      AN    OV;
      SAVE;
      CLR;
_005: A     BR;
      );
      JNB   _006;
      L     #REF_CUT_TAIL;
      L     #SPID_HMD;
      /R;
      T     #TIM_TEAL_2;
      AN    OV;
      SAVE;
      CLR;
_006: A     BR;
      );
      JNB   _007;
      L     #TIM_TEAL_1;
      L     #TIM_TEAL_2;
      -R;
      T     #TIM_TEAL_3;
_007: NOP   0;
NETWORK
TITLE =
      A(;
      L     #TIM_TEAL_3;
      L     0.000000e+00;
      ==R;
      );
      JNB   _008;
      L     1.000000e-04;
      T     #TIM_TEAL_3;
_008: NOP   0;
NETWORK
TITLE =
      L     #TIM_TEAL_3;
      L     #HW_TIM_SH;
      -R;
      T     #TIM_TEAL_ALL;
      NOP   0;
END_FUNCTION_BLOCK

FUNCTION FC 18 : VOID
AUTHOR : ES_MAP
NAME : TASK
VERSION : 0.0
BEGIN
// body was compiled from an SCL source; compiled code not shown
END_FUNCTION

FUNCTION FC 55 : VOID
AUTHOR : ES_MAP
NAME : GROUP
VERSION : 0.0
BEGIN
// body was compiled from an SCL source; compiled code not shown
END_FUNCTION

FUNCTION "A_IN" : VOID	// FC 402
TITLE = Analog input block
AUTHOR : SB5BRM11
FAMILY : TMBASE
NAME : A_IN
VERSION : 1.0
VAR_INPUT
  XE : WORD ;	//Input word
  MR_FIN : REAL ;	//Measuring range final
  MR_INI : REAL ;	//Measuring range initial
  VA_UP : INT ;	//Digits value abnormal upper
  VA_LOW : INT ;	//Digits value abnormal lower
  CODE { S7_string_0 := '0..+/4-20mA/1-5V'; S7_string_1 := 'Range - .... +' }: BOOL ;	//Type of input card
  EN_LIM { S7_string_0 := 'Y not limited'; S7_string_1 := 'Y limited' }: BOOL ;	//Limit output to measuring range
END_VAR
VAR_OUTPUT
  Y : REAL ;	//Output value
  QF : BOOL ;	//Value abnormal
END_VAR
VAR_TEMP
  DELTA : REAL ;	//MR_FIN - MR_INI
  Y_LOC : REAL ;	//Calculated output local
  XE_LOC : REAL ;	//Input transferred to local variable
  FACT : REAL ;
END_VAR
BEGIN
NETWORK
TITLE =
      SET;
      SAVE;
      =     L 16.1;
      L     #VA_UP;
      L     #VA_LOW;
      <I;
      L     #MR_FIN;
      L     #MR_INI;
      =     L 16.2;
      <R;
      O     L 16.2;
      JCN   A7d0;
      CLR;
      =     L 16.1;
      SAVE;
      BEU;
A7d0: L     #XE;
      ITD;
      DTR;
      T     #XE_LOC;
      CLR;
      A     #CODE;
      JCN   A7d1;
      L     #MR_FIN;
      L     5.529600e+04;
      /R;
      L     #MR_INI;
      TAK;
      T     LD 18;
      TAK;
      L     5.529600e+04;
      /R;
      L     LD 18;
      TAK;
      -R;
      T     #DELTA;
      L     #XE_LOC;
      *R;
      L     2.764800e+04;
      TAK;
      T     LD 18;
      TAK;
      L     #DELTA;
      *R;
      L     LD 18;
      +R;
      L     #MR_INI;
      +R;
      T     #Y_LOC;
      JU    A7d2;
A7d1: L     #MR_FIN;
      L     2.764800e+04;
      /R;
      L     #MR_INI;
      TAK;
      T     LD 18;
      TAK;
      L     2.764800e+04;
      /R;
      L     LD 18;
      TAK;
      -R;
      T     #DELTA;
      L     #XE_LOC;
      *R;
      L     #MR_INI;
      +R;
      T     #Y_LOC;
A7d2: CLR;
      A     #EN_LIM;
      JCN   A7d3;
      L     #Y_LOC;
      L     #MR_INI;
      <=R;
      JCN   A7d4;
      L     #MR_INI;
      T     #Y_LOC;
A7d4: L     #Y_LOC;
      L     #MR_FIN;
      >=R;
      JCN   A7d3;
      L     #MR_FIN;
      T     #Y_LOC;
A7d3: L     #XE;
      L     #VA_UP;
      >I;
      L     #XE;
      L     #VA_LOW;
      =     L 16.2;
      <I;
      O     L 16.2;
      =     #QF;
      L     #Y_LOC;
      T     #Y;
      A     L 16.1;
      SAVE;
      BE;
END_FUNCTION

FUNCTION "N_AW_BO" : VOID	// FC 430
VERSION : 0.1
VAR_INPUT
  IN1 : WORD ;
  IN2 : WORD ;
END_VAR
VAR_OUTPUT
  QRES : BOOL ;
END_VAR
VAR_TEMP
  Res : BOOL ;
END_VAR
BEGIN
NETWORK
TITLE =
      L     #IN1;
      L     #IN2;
      AW;
      L     0;
      <>I;
      =     #QRES;
END_FUNCTION

// DB 61: know-how protected block, not included

DATA_BLOCK DB 62
AUTHOR : ES_MAP
FAMILY : POOL
NAME : POOL
VERSION : 0.0
STRUCT
  POOL_bool : ARRAY[0..127] OF BOOL;
END_STRUCT;
BEGIN
   POOL_bool[0] := TRUE;
   POOL_bool[8] := TRUE;
   POOL_bool[10] := TRUE;
   POOL_bool[11] := TRUE;
   POOL_bool[13] := TRUE;
   POOL_bool[15] := TRUE;
   POOL_bool[17] := TRUE;
END_DATA_BLOCK

DATA_BLOCK DB 63
AUTHOR : ES_MAP
FAMILY : Projets
NAME : INSTANCE
VERSION : 0.0
"VISU_GEN"
BEGIN
END_DATA_BLOCK

DATA_BLOCK DB 64
AUTHOR : ES_MAP
FAMILY : Projects
NAME : INSTANCE
VERSION : 0.0
"READY_STD"
BEGIN
END_DATA_BLOCK

DATA_BLOCK DB 65
AUTHOR : ES_MAP
NAME : INSTANCE
VERSION : 0.0
"N_PID"
BEGIN
END_DATA_BLOCK

DATA_BLOCK DB 66
AUTHOR : ES_MAP
NAME : INSTANCE
VERSION : 0.0
"regulator"
BEGIN
END_DATA_BLOCK

DATA_BLOCK DB 67
AUTHOR : ES_MAP
FAMILY : IMPULS
NAME : INSTANCE
VERSION : 0.0
"TIMER_P"
BEGIN
END_DATA_BLOCK

DATA_BLOCK DB 68
AUTHOR : ES_MAP
FAMILY : IMPULS
NAME : INSTANCE
VERSION : 0.0
"TIMER_P"
BEGIN
END_DATA_BLOCK

DATA_BLOCK DB 69
AUTHOR : ES_MAP
NAME : INSTANCE
VERSION : 0.0
"CUT_SHER"
BEGIN
END_DATA_BLOCK

DATA_BLOCK DB 70
AUTHOR : ES_MAP
NAME : INSTANCE
VERSION : 0.0
"N_TOF"
BEGIN
END_DATA_BLOCK

DATA_BLOCK DB 72
AUTHOR : ES_MAP
NAME : INSTANCE
VERSION : 0.0
"N_AnMeas"
BEGIN
END_DATA_BLOCK

ORGANIZATION_BLOCK "CYCL_EXC"	// OB 1
TITLE = "Main Program Sweep (Cycle)"
VERSION : 0.1
VAR_TEMP
  OB1_EV_CLASS : BYTE ;	//Bits 0-3 = 1 (Coming event), Bits 4-7 = 1 (Event class 1)
  OB1_SCAN_1 : BYTE ;	//1 (Cold restart scan 1 of OB 1), 3 (Scan 2-n of OB 1)
  OB1_PRIORITY : BYTE ;	//Priority of OB Execution
  OB1_OB_NUMBR : BYTE ;	//1 (Organization block 1, OB1)
  OB1_RESERVED_1 : BYTE ;	//Reserved for system
  OB1_RESERVED_2 : BYTE ;	//Reserved for system
  OB1_PREV_CYCLE : INT ;	//Cycle time of previous OB1 scan (milliseconds)
  OB1_MIN_CYCLE : INT ;	//Minimum cycle time of OB1 (milliseconds)
  OB1_MAX_CYCLE : INT ;	//Maximum cycle time of OB1 (milliseconds)
  OB1_DATE_TIME : DATE_AND_TIME ;	//Date and time OB1 started
END_VAR
BEGIN
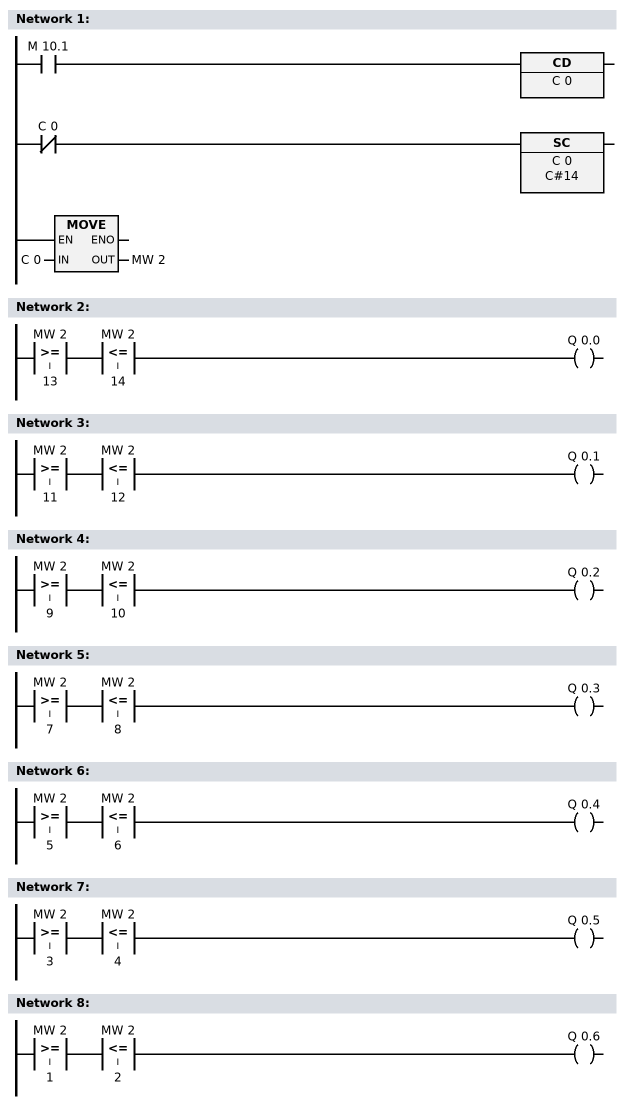
NETWORK
TITLE =
      A     M 10.1;
      CD    C 0;
      BLD   101;
      AN    C 0;
      L     C#14;
      S     C 0;
      NOP   0;
      L     C 0;
      T     MW 2;
      NOP   0;
      NOP   0;
NETWORK
TITLE =
      A(;
      L     MW 2;
      L     13;
      >=I;
      );
      A(;
      L     MW 2;
      L     14;
      <=I;
      );
      =     Q 0.0;
NETWORK
TITLE =
      A(;
      L     MW 2;
      L     11;
      >=I;
      );
      A(;
      L     MW 2;
      L     12;
      <=I;
      );
      =     Q 0.1;
NETWORK
TITLE =
      A(;
      L     MW 2;
      L     9;
      >=I;
      );
      A(;
      L     MW 2;
      L     10;
      <=I;
      );
      =     Q 0.2;
NETWORK
TITLE =
      A(;
      L     MW 2;
      L     7;
      >=I;
      );
      A(;
      L     MW 2;
      L     8;
      <=I;
      );
      =     Q 0.3;
NETWORK
TITLE =
      A(;
      L     MW 2;
      L     5;
      >=I;
      );
      A(;
      L     MW 2;
      L     6;
      <=I;
      );
      =     Q 0.4;
NETWORK
TITLE =
      A(;
      L     MW 2;
      L     3;
      >=I;
      );
      A(;
      L     MW 2;
      L     4;
      <=I;
      );
      =     Q 0.5;
NETWORK
TITLE =
      A(;
      L     MW 2;
      L     1;
      >=I;
      );
      A(;
      L     MW 2;
      L     2;
      <=I;
      );
      =     Q 0.6;
END_ORGANIZATION_BLOCK

ORGANIZATION_BLOCK OB 35
AUTHOR : ES_MAP
VERSION : 0.0
VAR_TEMP
  X : ARRAY  [1 .. 20 ] OF BYTE ;
END_VAR
BEGIN
// body was compiled from an SCL source; compiled code not shown
END_ORGANIZATION_BLOCK
